// Mitsubishi GX Works2 project: GLED-3K680-20090012_210325   PLC: FX3U/FX3UC
// SECS

PROGRAM MAIN
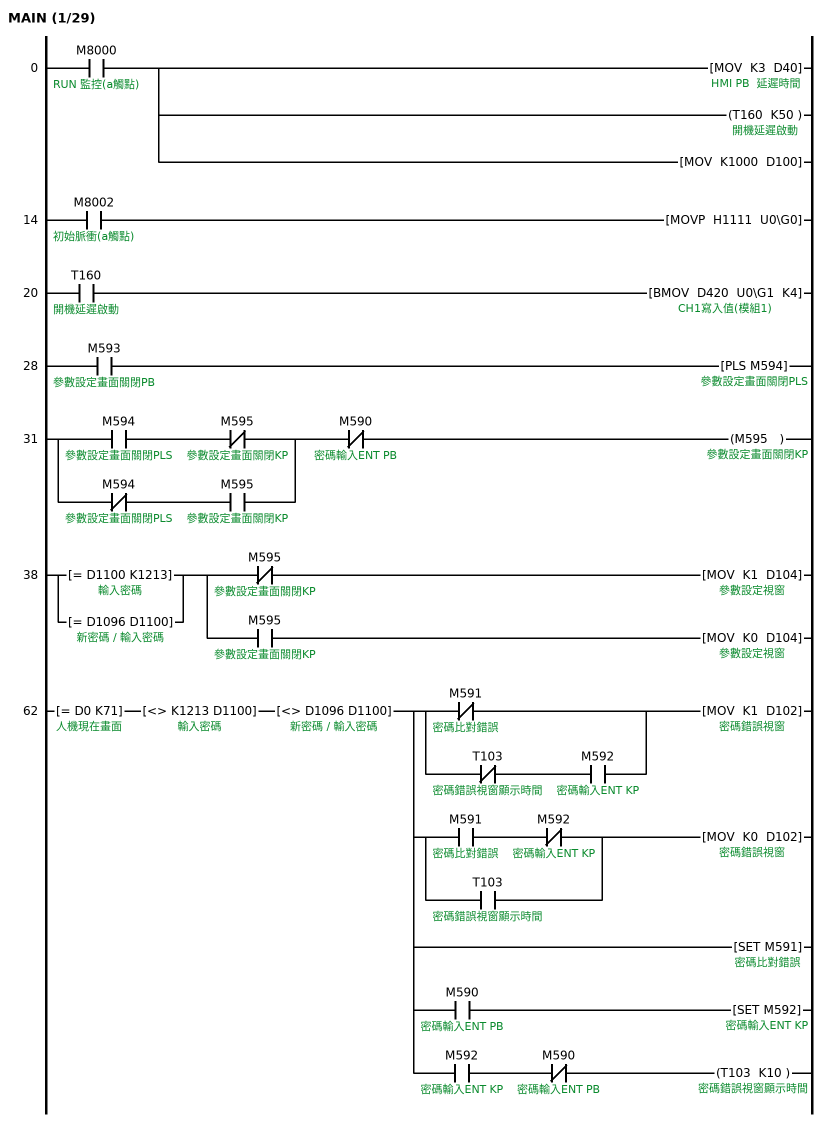
0     LD      M8000  ; RUN 監控(a觸點)
      MOV     K3 D40  ; HMI PB  延遲時間
      OUT     T160 K50  ; 開機延遲啟動
      MOV     K1000 D100
14    LD      M8002  ; 初始脈衝(a觸點)
      MOVP    H1111 U0\G0
20    LD      T160  ; 開機延遲啟動
      BMOV    D420 U0\G1 K4  ; CH1寫入值(模組1)
28    LD      M593  ; 參數設定畫面關閉PB
      PLS     M594  ; 參數設定畫面關閉PLS
31    LD      M594  ; 參數設定畫面關閉PLS
      ANI     M595  ; 參數設定畫面關閉KP
      LDI     M594  ; 參數設定畫面關閉PLS
      AND     M595  ; 參數設定畫面關閉KP
      ORB
      ANI     M590  ; 密碼輸入ENT PB
      OUT     M595  ; 參數設定畫面關閉KP
38    LD=     D1100 K1213  ; 輸入密碼
      OR=     D1096 D1100  ; 新密碼 / 輸入密碼
      MPS
      ANI     M595  ; 參數設定畫面關閉KP
      MOV     K1 D104  ; 參數設定視窗
      MPP
      AND     M595  ; 參數設定畫面關閉KP
      MOV     K0 D104
62    LD=     D0 K71  ; 人機現在畫面
      AND<>   K1213 D1100  ; 輸入密碼
      AND<>   D1096 D1100  ; 新密碼 / 輸入密碼
      MPS
      LDI     M591  ; 密碼比對錯誤
      LDI     T103  ; 密碼錯誤視窗顯示時間
      AND     M592  ; 密碼輸入ENT KP
      ORB
      ANB
      MOV     K1 D102  ; 密碼錯誤視窗
      MRD
      LD      M591  ; 密碼比對錯誤
      ANI     M592  ; 密碼輸入ENT KP
      OR      T103  ; 密碼錯誤視窗顯示時間
      ANB
      MOV     K0 D102
      MPP
      SET     M591  ; 密碼比對錯誤
      MPS
      AND     M590  ; 密碼輸入ENT PB
      SET     M592  ; 密碼輸入ENT KP
      MPP
      AND     M592  ; 密碼輸入ENT KP
      ANI     M590  ; 密碼輸入ENT PB
      OUT     T103 K10  ; 密碼錯誤視窗顯示時間
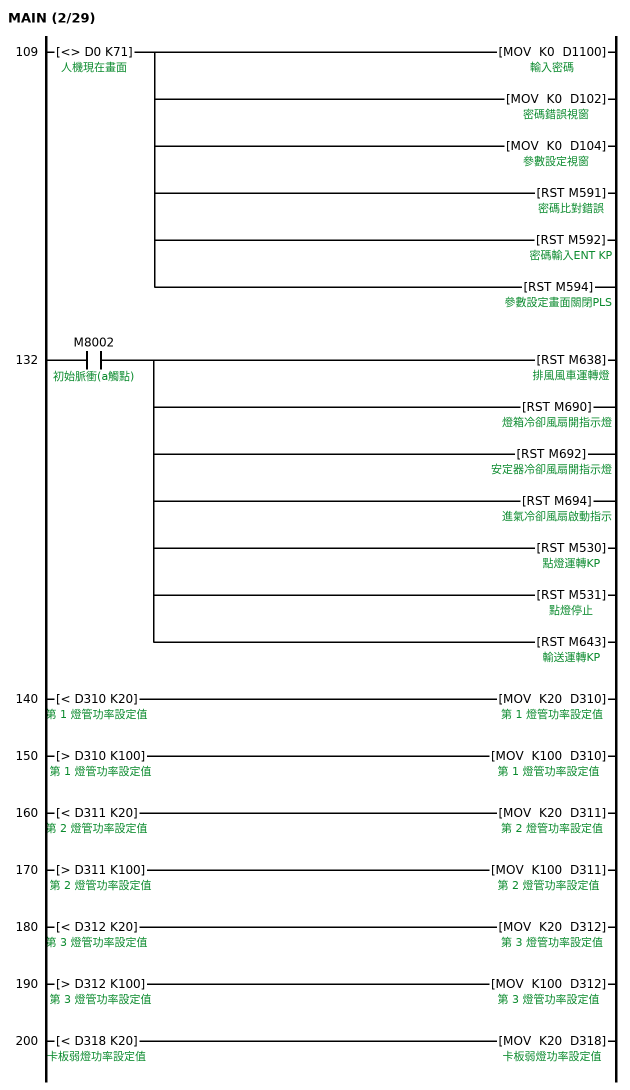
109   LD<>    D0 K71  ; 人機現在畫面
      MOV     K0 D1100
      MOV     K0 D102
      MOV     K0 D104
      RST     M591  ; 密碼比對錯誤
      RST     M592  ; 密碼輸入ENT KP
      RST     M594  ; 參數設定畫面關閉PLS
132   LD      M8002  ; 初始脈衝(a觸點)
      RST     M638  ; 排風風車運轉燈
      RST     M690  ; 燈箱冷卻風扇開指示燈
      RST     M692  ; 安定器冷卻風扇開指示燈
      RST     M694  ; 進氣冷卻風扇啟動指示
      RST     M530  ; 點燈運轉KP
      RST     M531  ; 點燈停止
      RST     M643  ; 輸送運轉KP
140   LD<     D310 K20  ; 第 1 燈管功率設定值
      MOV     K20 D310
150   LD>     D310 K100  ; 第 1 燈管功率設定值
      MOV     K100 D310
160   LD<     D311 K20  ; 第 2 燈管功率設定值
      MOV     K20 D311
170   LD>     D311 K100  ; 第 2 燈管功率設定值
      MOV     K100 D311
180   LD<     D312 K20  ; 第 3 燈管功率設定值
      MOV     K20 D312
190   LD>     D312 K100  ; 第 3 燈管功率設定值
      MOV     K100 D312
200   LD<     D318 K20  ; 卡板弱燈功率設定值
      MOV     K20 D318
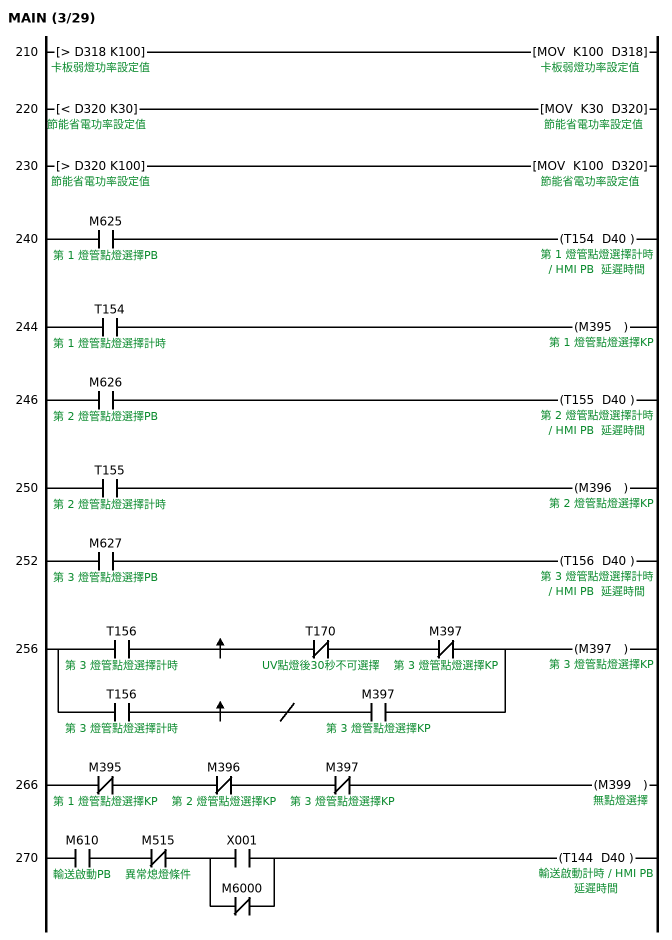
210   LD>     D318 K100  ; 卡板弱燈功率設定值
      MOV     K100 D318
220   LD<     D320 K30  ; 節能省電功率設定值
      MOV     K30 D320
230   LD>     D320 K100  ; 節能省電功率設定值
      MOV     K100 D320
240   LD      M625  ; 第 1 燈管點燈選擇PB
      OUT     T154 D40  ; 第 1 燈管點燈選擇計時 / HMI PB  延遲時間
244   LD      T154  ; 第 1 燈管點燈選擇計時
      OUT     M395  ; 第 1 燈管點燈選擇KP
246   LD      M626  ; 第 2 燈管點燈選擇PB
      OUT     T155 D40  ; 第 2 燈管點燈選擇計時 / HMI PB  延遲時間
250   LD      T155  ; 第 2 燈管點燈選擇計時
      OUT     M396  ; 第 2 燈管點燈選擇KP
252   LD      M627  ; 第 3 燈管點燈選擇PB
      OUT     T156 D40  ; 第 3 燈管點燈選擇計時 / HMI PB  延遲時間
256   LD      T156  ; 第 3 燈管點燈選擇計時
      MEP
      ANI     T170  ; UV點燈後30秒不可選擇
      ANI     M397  ; 第 3 燈管點燈選擇KP
      LD      T156  ; 第 3 燈管點燈選擇計時
      MEP
      INV
      AND     M397  ; 第 3 燈管點燈選擇KP
      ORB
      OUT     M397  ; 第 3 燈管點燈選擇KP
266   LDI     M395  ; 第 1 燈管點燈選擇KP
      ANI     M396  ; 第 2 燈管點燈選擇KP
      ANI     M397  ; 第 3 燈管點燈選擇KP
      OUT     M399  ; 無點燈選擇
270   LD      M610  ; 輸送啟動PB
      ANI     M515  ; 異常熄燈條件
      LD      X001
      ORI     M6000
      ANB
      OUT     T144 D40  ; 輸送啟動計時 / HMI PB  延遲時間
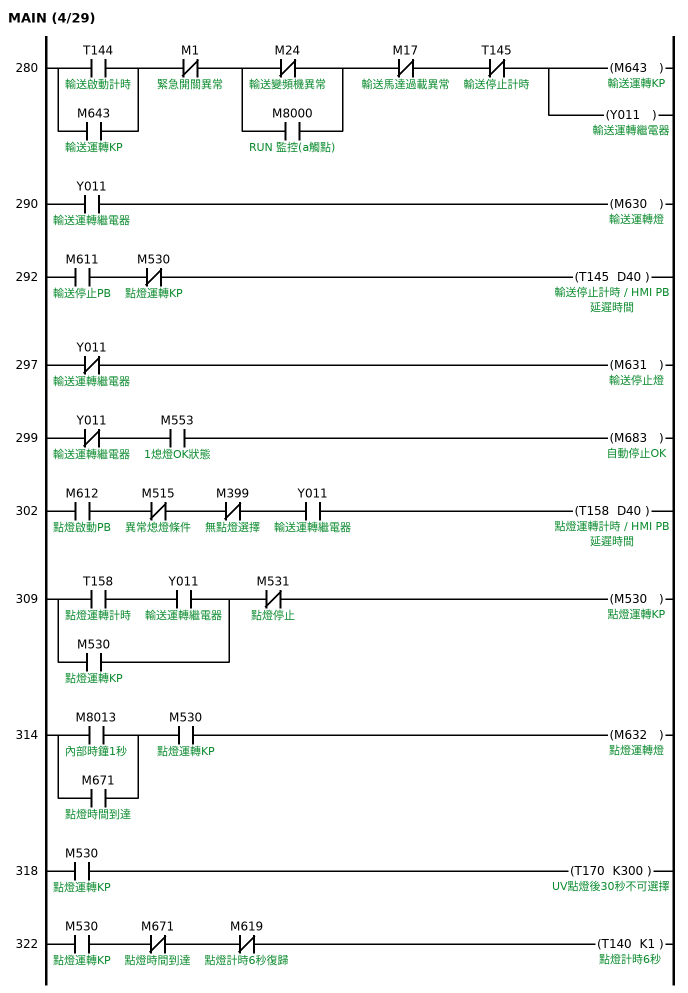
280   LD      T144  ; 輸送啟動計時
      OR      M643  ; 輸送運轉KP
      ANI     M1  ; 緊急開關異常
      LDI     M24  ; 輸送變頻機異常
      OR      M8000  ; RUN 監控(a觸點)
      ANB
      ANI     M17  ; 輸送馬達過載異常
      ANI     T145  ; 輸送停止計時
      OUT     M643  ; 輸送運轉KP
      OUT     Y011  ; 輸送運轉繼電器
290   LD      Y011  ; 輸送運轉繼電器
      OUT     M630  ; 輸送運轉燈
292   LD      M611  ; 輸送停止PB
      ANI     M530  ; 點燈運轉KP
      OUT     T145 D40  ; 輸送停止計時 / HMI PB  延遲時間
297   LDI     Y011  ; 輸送運轉繼電器
      OUT     M631  ; 輸送停止燈
299   LDI     Y011  ; 輸送運轉繼電器
      AND     M553  ; 1熄燈OK狀態
      OUT     M683  ; 自動停止OK
302   LD      M612  ; 點燈啟動PB
      ANI     M515  ; 異常熄燈條件
      ANI     M399  ; 無點燈選擇
      AND     Y011  ; 輸送運轉繼電器
      OUT     T158 D40  ; 點燈運轉計時 / HMI PB  延遲時間
309   LD      T158  ; 點燈運轉計時
      AND     Y011  ; 輸送運轉繼電器
      OR      M530  ; 點燈運轉KP
      ANI     M531  ; 點燈停止
      OUT     M530  ; 點燈運轉KP
314   LD      M8013  ; 內部時鐘1秒
      OR      M671  ; 點燈時間到達
      AND     M530  ; 點燈運轉KP
      OUT     M632  ; 點燈運轉燈
318   LD      M530  ; 點燈運轉KP
      OUT     T170 K300  ; UV點燈後30秒不可選擇
322   LD      M530  ; 點燈運轉KP
      ANI     M671  ; 點燈時間到達
      ANI     M619  ; 點燈計時6秒復歸
      OUT     T140 K1  ; 點燈計時6秒
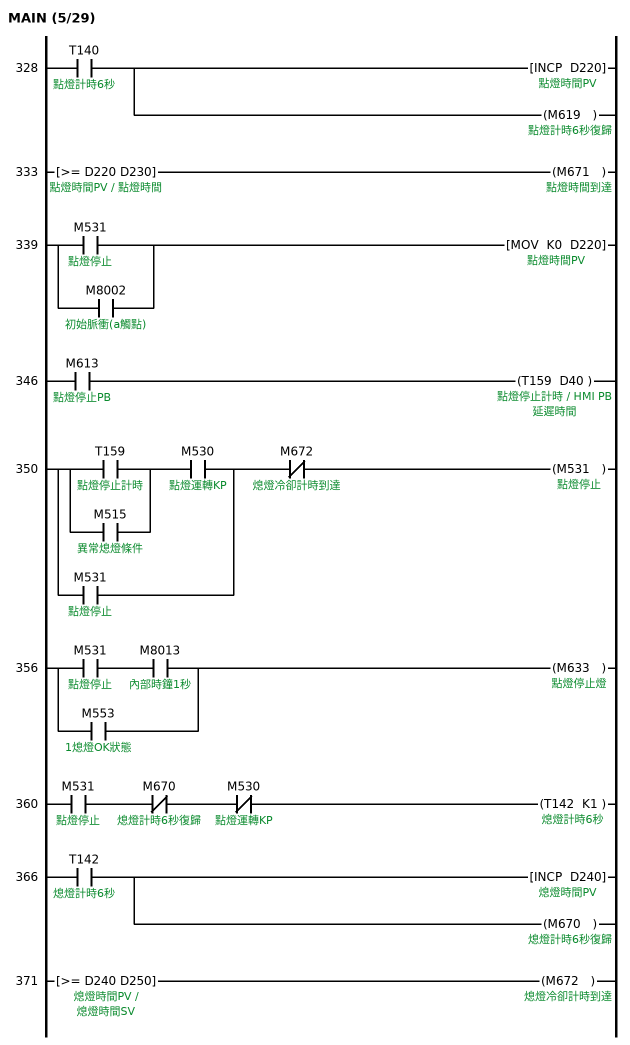
328   LD      T140  ; 點燈計時6秒
      INCP    D220  ; 點燈時間PV
      OUT     M619  ; 點燈計時6秒復歸
333   LD>=    D220 D230  ; 點燈時間PV / 點燈時間
      OUT     M671  ; 點燈時間到達
339   LD      M531  ; 點燈停止
      OR      M8002  ; 初始脈衝(a觸點)
      MOV     K0 D220
346   LD      M613  ; 點燈停止PB
      OUT     T159 D40  ; 點燈停止計時 / HMI PB  延遲時間
350   LD      T159  ; 點燈停止計時
      OR      M515  ; 異常熄燈條件
      AND     M530  ; 點燈運轉KP
      OR      M531  ; 點燈停止
      ANI     M672  ; 熄燈冷卻計時到達
      OUT     M531  ; 點燈停止
356   LD      M531  ; 點燈停止
      AND     M8013  ; 內部時鐘1秒
      OR      M553  ; 1熄燈OK狀態
      OUT     M633  ; 點燈停止燈
360   LD      M531  ; 點燈停止
      ANI     M670  ; 熄燈計時6秒復歸
      ANI     M530  ; 點燈運轉KP
      OUT     T142 K1  ; 熄燈計時6秒
366   LD      T142  ; 熄燈計時6秒
      INCP    D240  ; 熄燈時間PV
      OUT     M670  ; 熄燈計時6秒復歸
371   LD>=    D240 D250  ; 熄燈時間PV / 熄燈時間SV
      OUT     M672  ; 熄燈冷卻計時到達
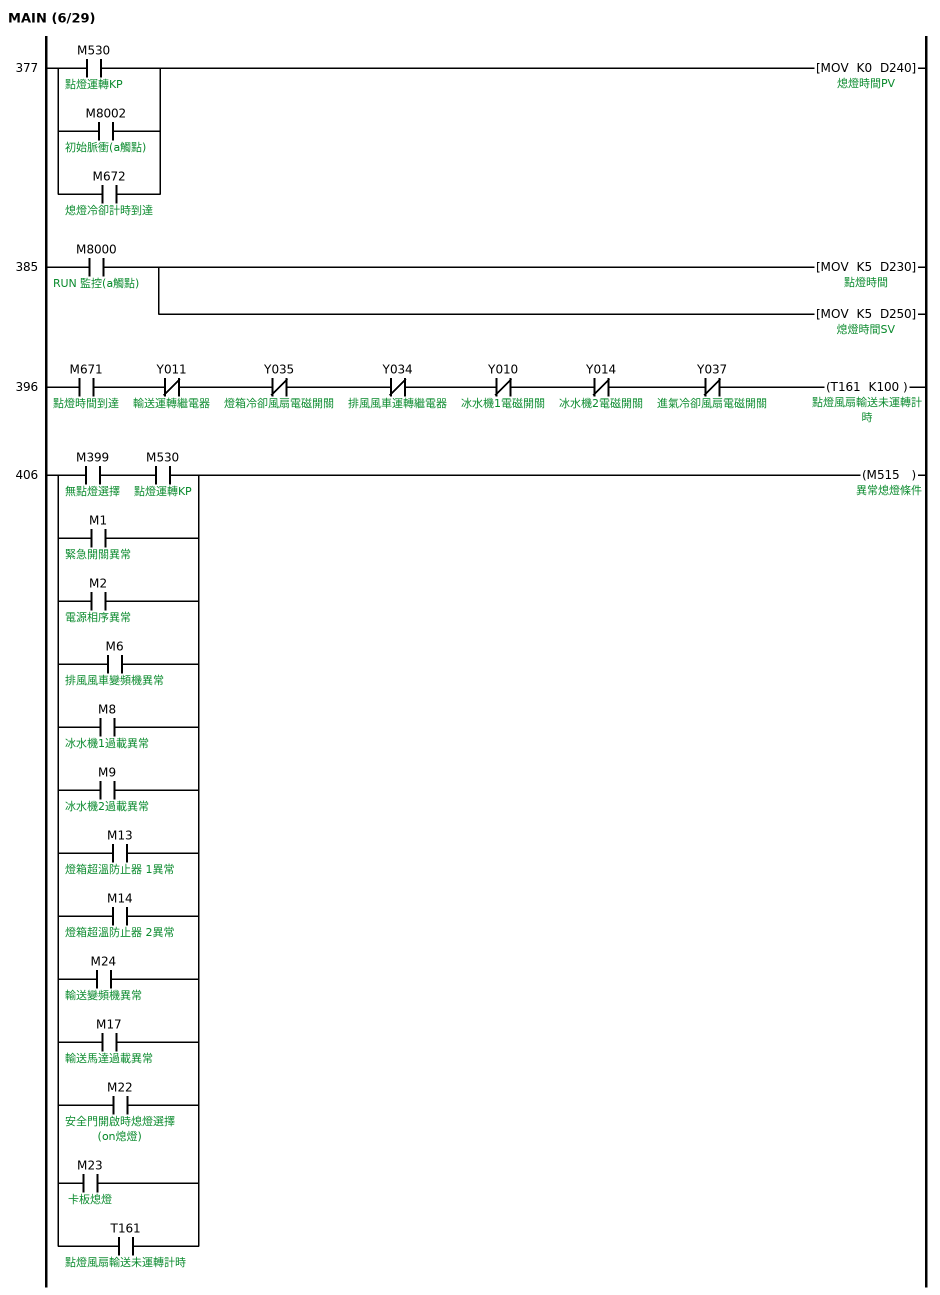
377   LD      M530  ; 點燈運轉KP
      OR      M8002  ; 初始脈衝(a觸點)
      OR      M672  ; 熄燈冷卻計時到達
      MOV     K0 D240
385   LD      M8000  ; RUN 監控(a觸點)
      MOV     K5 D230
      MOV     K5 D250
396   LD      M671  ; 點燈時間到達
      ANI     Y011  ; 輸送運轉繼電器
      ANI     Y035  ; 燈箱冷卻風扇電磁開關
      ANI     Y034  ; 排風風車運轉繼電器
      ANI     Y010  ; 冰水機1電磁開關
      ANI     Y014  ; 冰水機2電磁開關
      ANI     Y037  ; 進氣冷卻風扇電磁開關
      OUT     T161 K100  ; 點燈風扇輸送未運轉計時
406   LD      M399  ; 無點燈選擇
      AND     M530  ; 點燈運轉KP
      OR      M1  ; 緊急開關異常
      OR      M2  ; 電源相序異常
      OR      M6  ; 排風風車變頻機異常
      OR      M8  ; 冰水機1過載異常
      OR      M9  ; 冰水機2過載異常
      OR      M13  ; 燈箱超溫防止器 1異常
      OR      M14  ; 燈箱超溫防止器 2異常
      OR      M24  ; 輸送變頻機異常
      OR      M17  ; 輸送馬達過載異常
      OR      M22  ; 安全門開啟時熄燈選擇    (on熄燈)
      OR      M23  ; 卡板熄燈
      OR      T161  ; 點燈風扇輸送未運轉計時
      OUT     M515  ; 異常熄燈條件
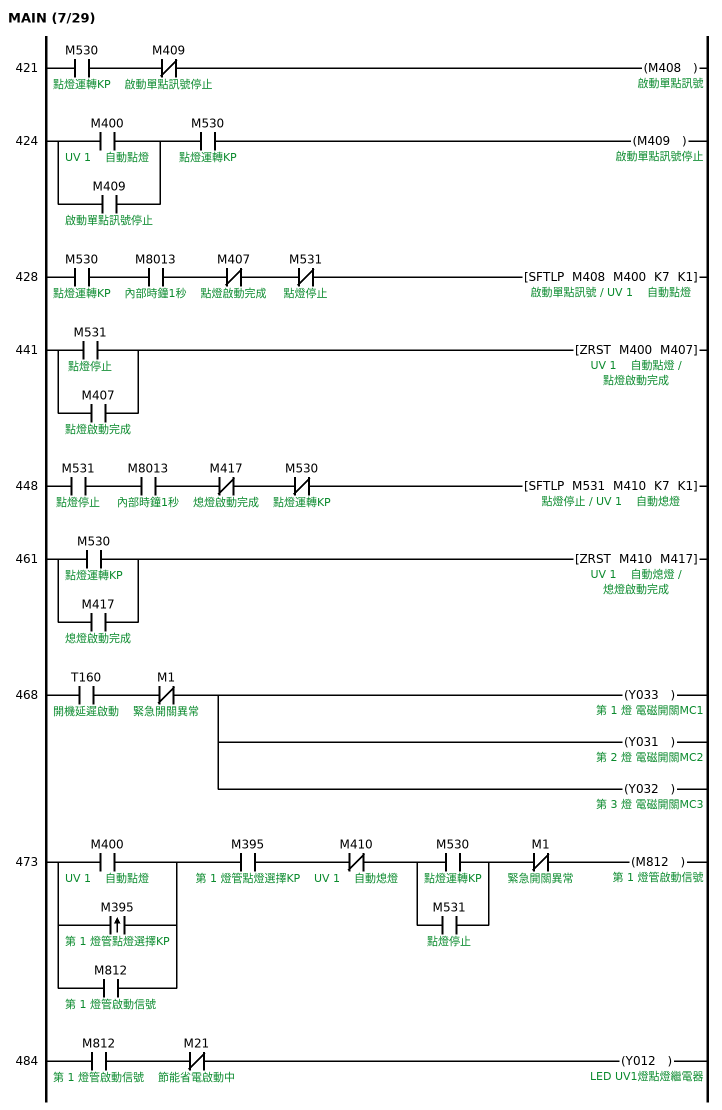
421   LD      M530  ; 點燈運轉KP
      ANI     M409  ; 啟動單點訊號停止
      OUT     M408  ; 啟動單點訊號
424   LD      M400  ; UV 1    自動點燈
      OR      M409  ; 啟動單點訊號停止
      AND     M530  ; 點燈運轉KP
      OUT     M409  ; 啟動單點訊號停止
428   LD      M530  ; 點燈運轉KP
      AND     M8013  ; 內部時鐘1秒
      ANI     M407  ; 點燈啟動完成
      ANI     M531  ; 點燈停止
      SFTLP   M408 M400 K7 K1
441   LD      M531  ; 點燈停止
      OR      M407  ; 點燈啟動完成
      ZRST    M400 M407
448   LD      M531  ; 點燈停止
      AND     M8013  ; 內部時鐘1秒
      ANI     M417  ; 熄燈啟動完成
      ANI     M530  ; 點燈運轉KP
      SFTLP   M531 M410 K7 K1  ; UV 1    自動熄燈
461   LD      M530  ; 點燈運轉KP
      OR      M417  ; 熄燈啟動完成
      ZRST    M410 M417
468   LD      T160  ; 開機延遲啟動
      ANI     M1  ; 緊急開關異常
      OUT     Y033  ; 第 1 燈 電磁開關MC1
      OUT     Y031  ; 第 2 燈 電磁開關MC2
      OUT     Y032  ; 第 3 燈 電磁開關MC3
473   LD      M400  ; UV 1    自動點燈
      ORP     M395  ; 第 1 燈管點燈選擇KP
      OR      M812  ; 第 1 燈管啟動信號
      AND     M395  ; 第 1 燈管點燈選擇KP
      ANI     M410  ; UV 1    自動熄燈
      LD      M530  ; 點燈運轉KP
      OR      M531  ; 點燈停止
      ANB
      ANI     M1  ; 緊急開關異常
      OUT     M812  ; 第 1 燈管啟動信號
484   LD      M812  ; 第 1 燈管啟動信號
      ANI     M21  ; 節能省電啟動中
      OUT     Y012  ; LED UV1燈點燈繼電器
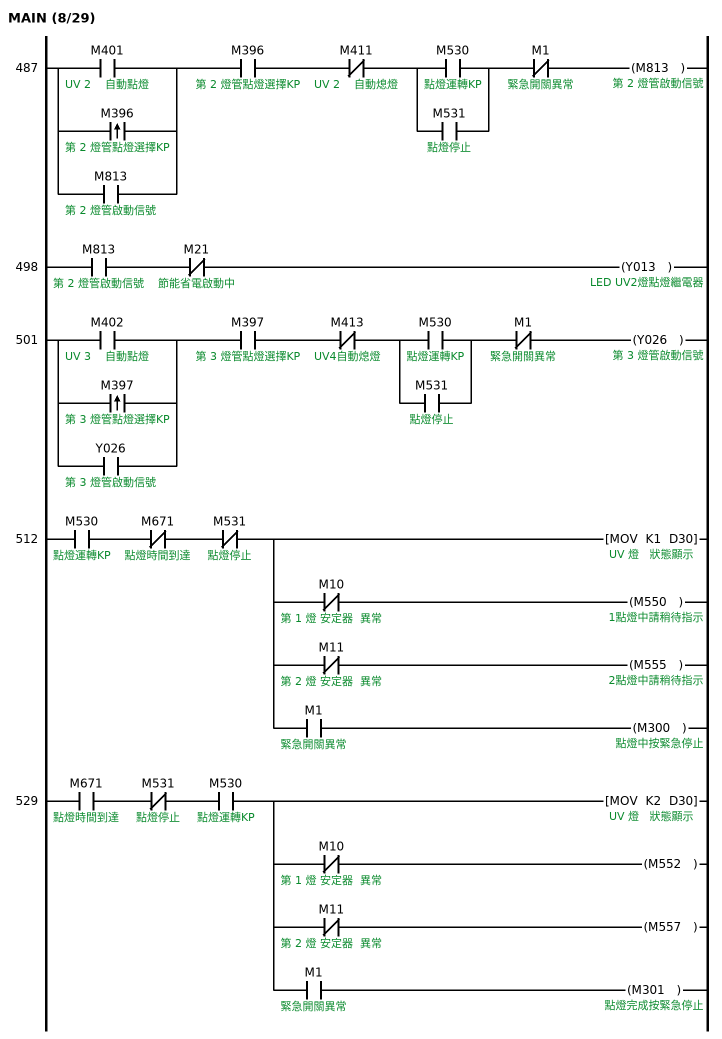
487   LD      M401  ; UV 2    自動點燈
      ORP     M396  ; 第 2 燈管點燈選擇KP
      OR      M813  ; 第 2 燈管啟動信號
      AND     M396  ; 第 2 燈管點燈選擇KP
      ANI     M411  ; UV 2    自動熄燈
      LD      M530  ; 點燈運轉KP
      OR      M531  ; 點燈停止
      ANB
      ANI     M1  ; 緊急開關異常
      OUT     M813  ; 第 2 燈管啟動信號
498   LD      M813  ; 第 2 燈管啟動信號
      ANI     M21  ; 節能省電啟動中
      OUT     Y013  ; LED UV2燈點燈繼電器
501   LD      M402  ; UV 3    自動點燈
      ORP     M397  ; 第 3 燈管點燈選擇KP
      OR      Y026  ; 第 3 燈管啟動信號
      AND     M397  ; 第 3 燈管點燈選擇KP
      ANI     M413  ; UV4自動熄燈
      LD      M530  ; 點燈運轉KP
      OR      M531  ; 點燈停止
      ANB
      ANI     M1  ; 緊急開關異常
      OUT     Y026  ; 第 3 燈管啟動信號
512   LD      M530  ; 點燈運轉KP
      ANI     M671  ; 點燈時間到達
      ANI     M531  ; 點燈停止
      MOV     K1 D30  ; UV 燈   狀態顯示
      MPS
      ANI     M10  ; 第 1 燈 安定器  異常
      OUT     M550  ; 1點燈中請稍待指示
      MRD
      ANI     M11  ; 第 2 燈 安定器  異常
      OUT     M555  ; 2點燈中請稍待指示
      MPP
      AND     M1  ; 緊急開關異常
      OUT     M300  ; 點燈中按緊急停止
529   LD      M671  ; 點燈時間到達
      ANI     M531  ; 點燈停止
      AND     M530  ; 點燈運轉KP
      MOV     K2 D30
      MPS
      ANI     M10  ; 第 1 燈 安定器  異常
      OUT     M552
      MRD
      ANI     M11  ; 第 2 燈 安定器  異常
      OUT     M557
      MPP
      AND     M1  ; 緊急開關異常
      OUT     M301  ; 點燈完成按緊急停止
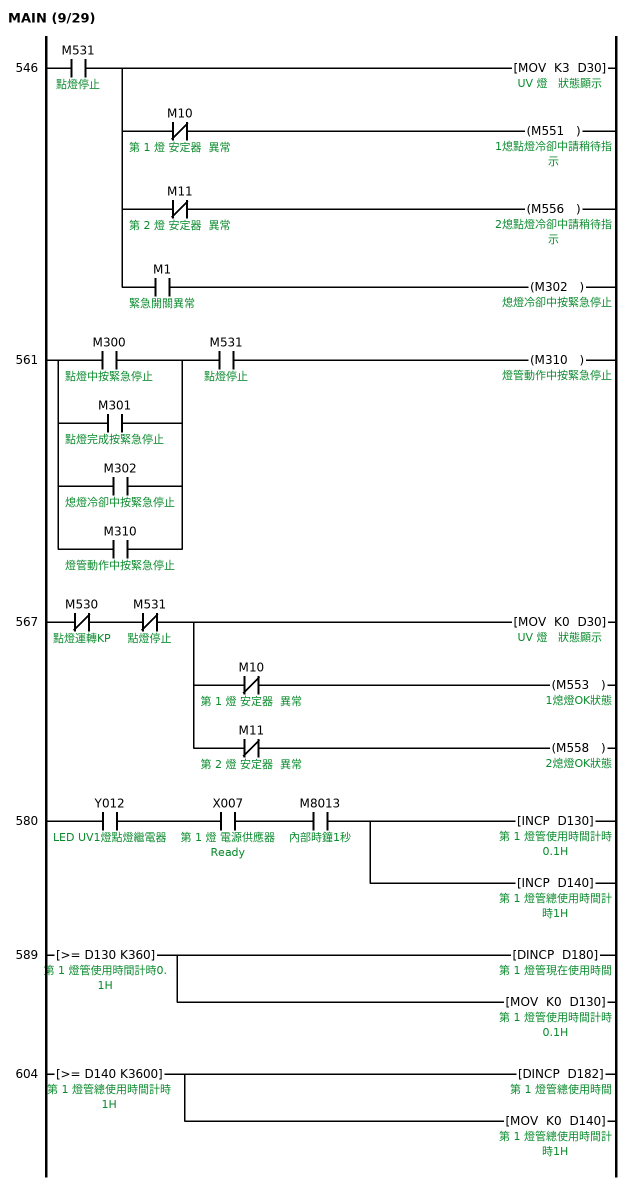
546   LD      M531  ; 點燈停止
      MOV     K3 D30
      MPS
      ANI     M10  ; 第 1 燈 安定器  異常
      OUT     M551  ; 1熄點燈冷卻中請稍待指示
      MRD
      ANI     M11  ; 第 2 燈 安定器  異常
      OUT     M556  ; 2熄點燈冷卻中請稍待指示
      MPP
      AND     M1  ; 緊急開關異常
      OUT     M302  ; 熄燈冷卻中按緊急停止
561   LD      M300  ; 點燈中按緊急停止
      OR      M301  ; 點燈完成按緊急停止
      OR      M302  ; 熄燈冷卻中按緊急停止
      OR      M310  ; 燈管動作中按緊急停止
      AND     M531  ; 點燈停止
      OUT     M310  ; 燈管動作中按緊急停止
567   LDI     M530  ; 點燈運轉KP
      ANI     M531  ; 點燈停止
      MOV     K0 D30
      MPS
      ANI     M10  ; 第 1 燈 安定器  異常
      OUT     M553  ; 1熄燈OK狀態
      MPP
      ANI     M11  ; 第 2 燈 安定器  異常
      OUT     M558  ; 2熄燈OK狀態
580   LD      Y012  ; LED UV1燈點燈繼電器
      AND     X007  ; 第 1 燈 電源供應器 Ready
      AND     M8013  ; 內部時鐘1秒
      INCP    D130  ; 第 1 燈管使用時間計時0.1H
      INCP    D140  ; 第 1 燈管總使用時間計時1H
589   LD>=    D130 K360  ; 第 1 燈管使用時間計時0.1H
      DINCP   D180  ; 第 1 燈管現在使用時間
      MOV     K0 D130
604   LD>=    D140 K3600  ; 第 1 燈管總使用時間計時1H
      DINCP   D182  ; 第 1 燈管總使用時間
      MOV     K0 D140
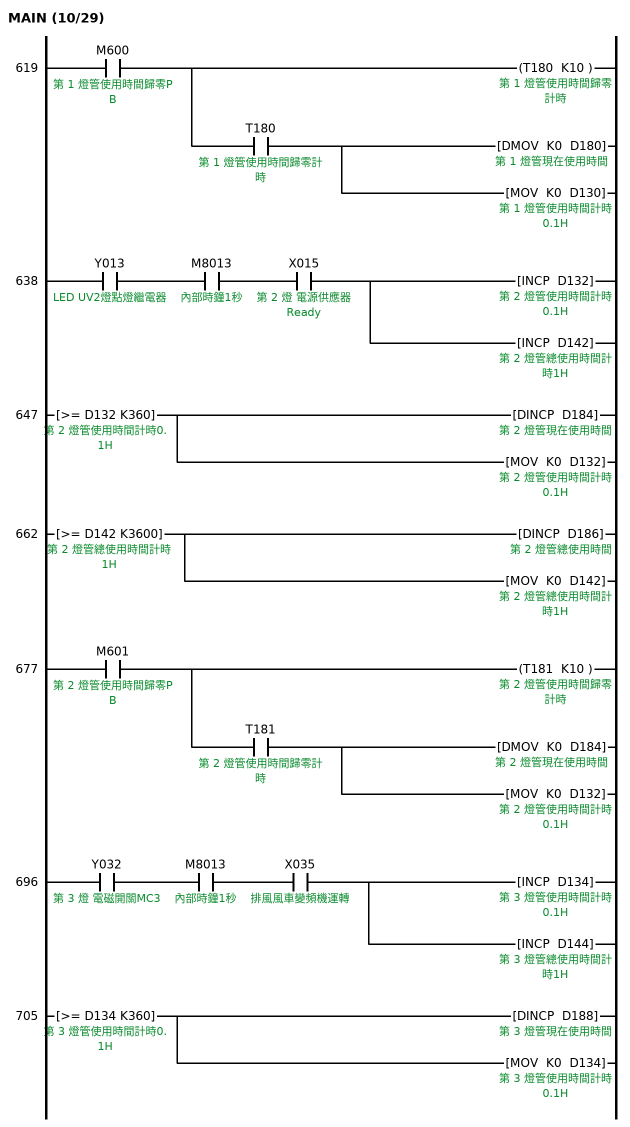
619   LD      M600  ; 第 1 燈管使用時間歸零PB
      OUT     T180 K10  ; 第 1 燈管使用時間歸零計時
      AND     T180  ; 第 1 燈管使用時間歸零計時
      DMOV    K0 D180
      MOV     K0 D130
638   LD      Y013  ; LED UV2燈點燈繼電器
      AND     M8013  ; 內部時鐘1秒
      AND     X015  ; 第 2 燈 電源供應器 Ready
      INCP    D132  ; 第 2 燈管使用時間計時0.1H
      INCP    D142  ; 第 2 燈管總使用時間計時1H
647   LD>=    D132 K360  ; 第 2 燈管使用時間計時0.1H
      DINCP   D184  ; 第 2 燈管現在使用時間
      MOV     K0 D132
662   LD>=    D142 K3600  ; 第 2 燈管總使用時間計時1H
      DINCP   D186  ; 第 2 燈管總使用時間
      MOV     K0 D142
677   LD      M601  ; 第 2 燈管使用時間歸零PB
      OUT     T181 K10  ; 第 2 燈管使用時間歸零計時
      AND     T181  ; 第 2 燈管使用時間歸零計時
      DMOV    K0 D184
      MOV     K0 D132
696   LD      Y032  ; 第 3 燈 電磁開關MC3
      AND     M8013  ; 內部時鐘1秒
      AND     X035  ; 排風風車變頻機運轉
      INCP    D134  ; 第 3 燈管使用時間計時0.1H
      INCP    D144  ; 第 3 燈管總使用時間計時1H
705   LD>=    D134 K360  ; 第 3 燈管使用時間計時0.1H
      DINCP   D188  ; 第 3 燈管現在使用時間
      MOV     K0 D134
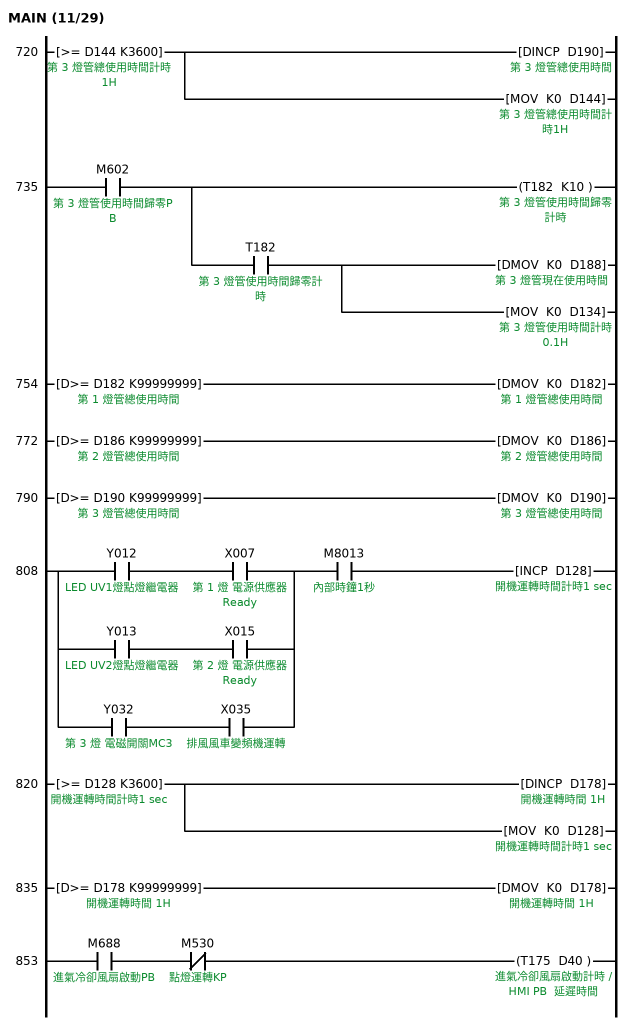
720   LD>=    D144 K3600  ; 第 3 燈管總使用時間計時1H
      DINCP   D190  ; 第 3 燈管總使用時間
      MOV     K0 D144
735   LD      M602  ; 第 3 燈管使用時間歸零PB
      OUT     T182 K10  ; 第 3 燈管使用時間歸零計時
      AND     T182  ; 第 3 燈管使用時間歸零計時
      DMOV    K0 D188
      MOV     K0 D134
754   LDD>=   D182 K99999999  ; 第 1 燈管總使用時間
      DMOV    K0 D182
772   LDD>=   D186 K99999999  ; 第 2 燈管總使用時間
      DMOV    K0 D186
790   LDD>=   D190 K99999999  ; 第 3 燈管總使用時間
      DMOV    K0 D190
808   LD      Y012  ; LED UV1燈點燈繼電器
      AND     X007  ; 第 1 燈 電源供應器 Ready
      LD      Y013  ; LED UV2燈點燈繼電器
      AND     X015  ; 第 2 燈 電源供應器 Ready
      ORB
      LD      Y032  ; 第 3 燈 電磁開關MC3
      AND     X035  ; 排風風車變頻機運轉
      ORB
      AND     M8013  ; 內部時鐘1秒
      INCP    D128  ; 開機運轉時間計時1 sec
820   LD>=    D128 K3600  ; 開機運轉時間計時1 sec
      DINCP   D178  ; 開機運轉時間 1H
      MOV     K0 D128
835   LDD>=   D178 K99999999  ; 開機運轉時間 1H
      DMOV    K0 D178
853   LD      M688  ; 進氣冷卻風扇啟動PB
      ANI     M530  ; 點燈運轉KP
      OUT     T175 D40  ; 進氣冷卻風扇啟動計時 / HMI PB  延遲時間
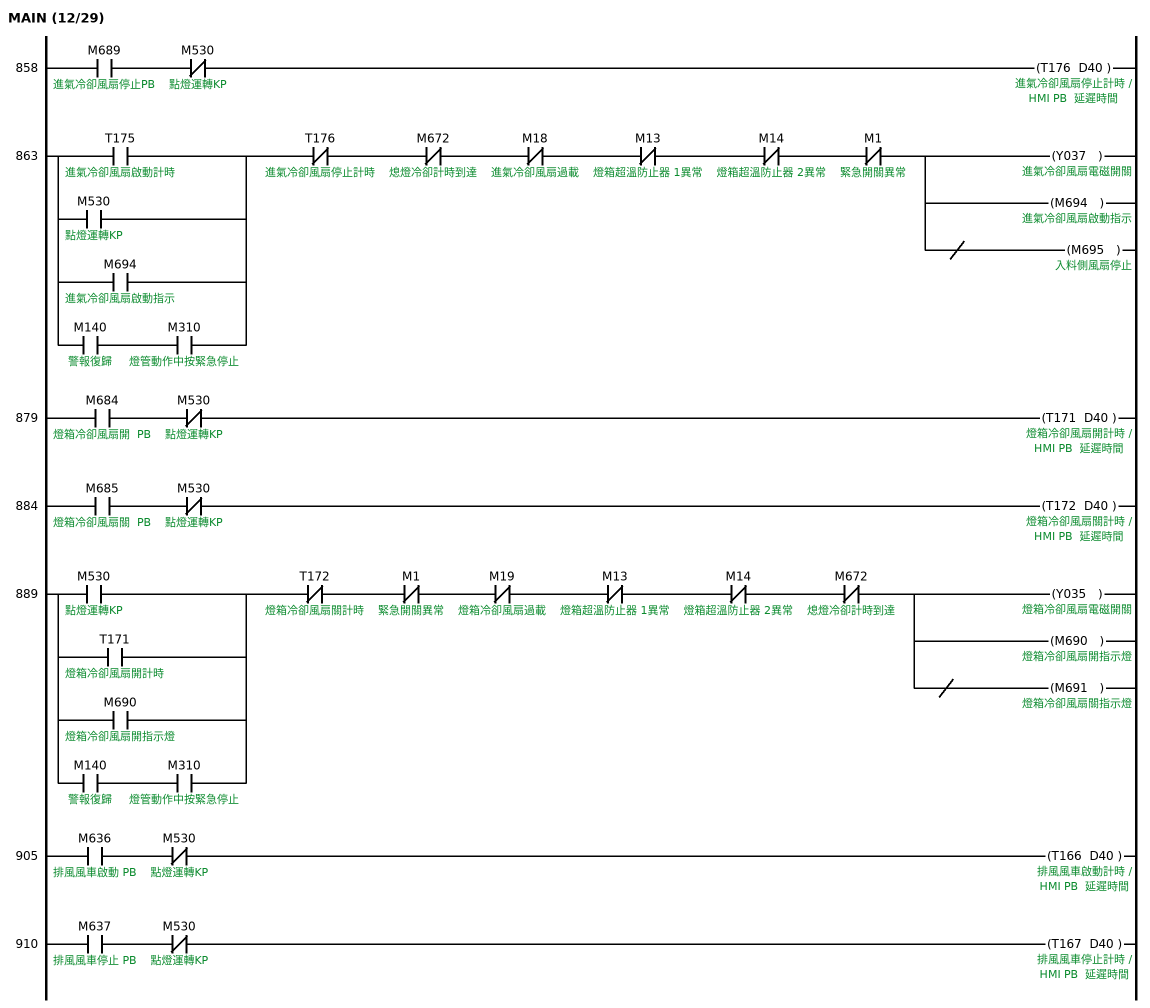
858   LD      M689  ; 進氣冷卻風扇停止PB
      ANI     M530  ; 點燈運轉KP
      OUT     T176 D40  ; 進氣冷卻風扇停止計時 / HMI PB  延遲時間
863   LD      T175  ; 進氣冷卻風扇啟動計時
      OR      M530  ; 點燈運轉KP
      OR      M694  ; 進氣冷卻風扇啟動指示
      LD      M140  ; 警報復歸
      AND     M310  ; 燈管動作中按緊急停止
      ORB
      ANI     T176  ; 進氣冷卻風扇停止計時
      ANI     M672  ; 熄燈冷卻計時到達
      ANI     M18  ; 進氣冷卻風扇過載
      ANI     M13  ; 燈箱超溫防止器 1異常
      ANI     M14  ; 燈箱超溫防止器 2異常
      ANI     M1  ; 緊急開關異常
      OUT     Y037  ; 進氣冷卻風扇電磁開關
      OUT     M694  ; 進氣冷卻風扇啟動指示
      INV
      OUT     M695  ; 入料側風扇停止
879   LD      M684  ; 燈箱冷卻風扇開  PB
      ANI     M530  ; 點燈運轉KP
      OUT     T171 D40  ; 燈箱冷卻風扇開計時 / HMI PB  延遲時間
884   LD      M685  ; 燈箱冷卻風扇關  PB
      ANI     M530  ; 點燈運轉KP
      OUT     T172 D40  ; 燈箱冷卻風扇關計時 / HMI PB  延遲時間
889   LD      M530  ; 點燈運轉KP
      OR      T171  ; 燈箱冷卻風扇開計時
      OR      M690  ; 燈箱冷卻風扇開指示燈
      LD      M140  ; 警報復歸
      AND     M310  ; 燈管動作中按緊急停止
      ORB
      ANI     T172  ; 燈箱冷卻風扇關計時
      ANI     M1  ; 緊急開關異常
      ANI     M19  ; 燈箱冷卻風扇過載
      ANI     M13  ; 燈箱超溫防止器 1異常
      ANI     M14  ; 燈箱超溫防止器 2異常
      ANI     M672  ; 熄燈冷卻計時到達
      OUT     Y035  ; 燈箱冷卻風扇電磁開關
      OUT     M690  ; 燈箱冷卻風扇開指示燈
      INV
      OUT     M691  ; 燈箱冷卻風扇關指示燈
905   LD      M636  ; 排風風車啟動 PB
      ANI     M530  ; 點燈運轉KP
      OUT     T166 D40  ; 排風風車啟動計時 / HMI PB  延遲時間
910   LD      M637  ; 排風風車停止 PB
      ANI     M530  ; 點燈運轉KP
      OUT     T167 D40  ; 排風風車停止計時 / HMI PB  延遲時間
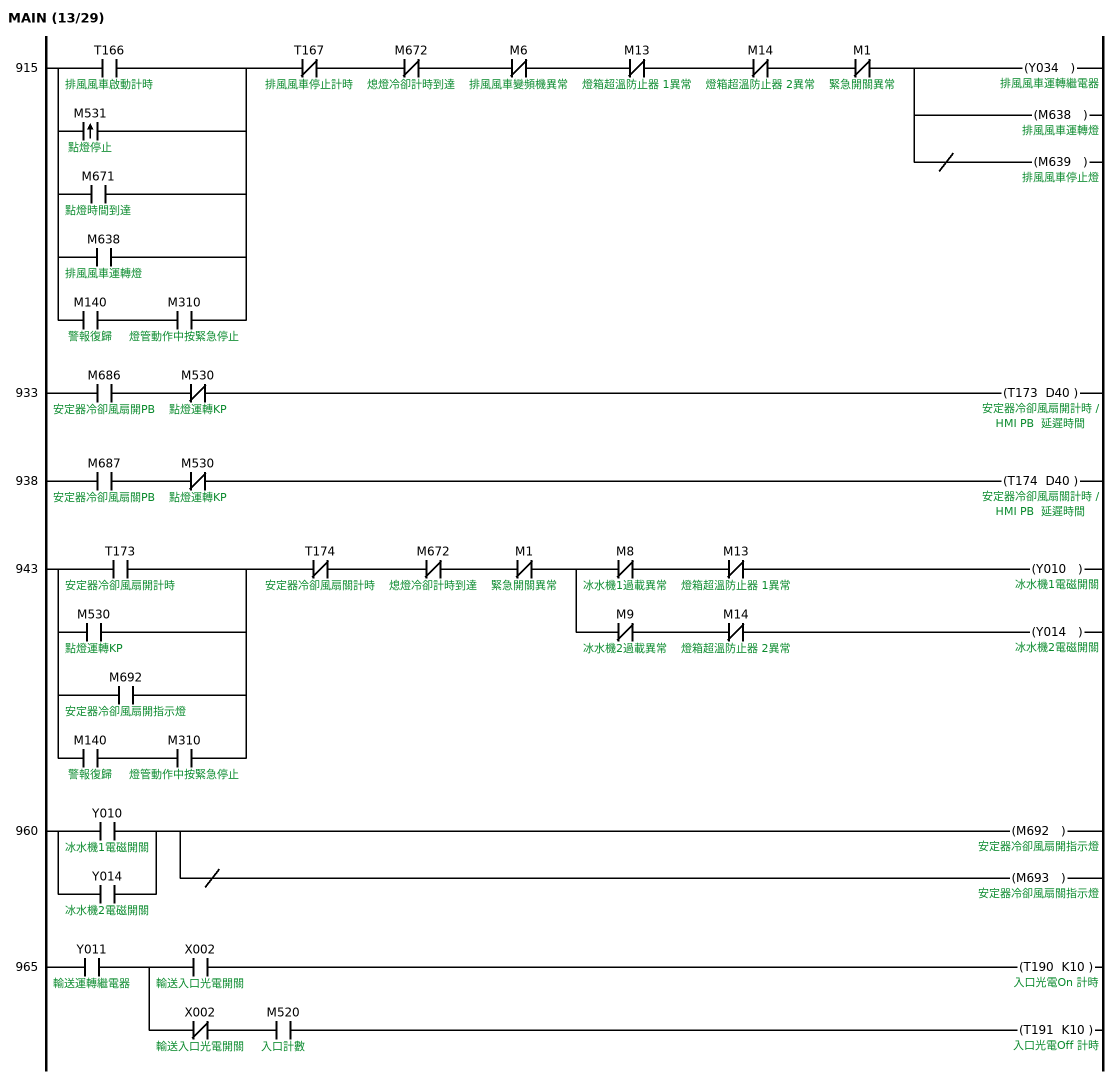
915   LD      T166  ; 排風風車啟動計時
      ORP     M531  ; 點燈停止
      OR      M671  ; 點燈時間到達
      OR      M638  ; 排風風車運轉燈
      LD      M140  ; 警報復歸
      AND     M310  ; 燈管動作中按緊急停止
      ORB
      ANI     T167  ; 排風風車停止計時
      ANI     M672  ; 熄燈冷卻計時到達
      ANI     M6  ; 排風風車變頻機異常
      ANI     M13  ; 燈箱超溫防止器 1異常
      ANI     M14  ; 燈箱超溫防止器 2異常
      ANI     M1  ; 緊急開關異常
      OUT     Y034  ; 排風風車運轉繼電器
      OUT     M638  ; 排風風車運轉燈
      INV
      OUT     M639  ; 排風風車停止燈
933   LD      M686  ; 安定器冷卻風扇開PB
      ANI     M530  ; 點燈運轉KP
      OUT     T173 D40  ; 安定器冷卻風扇開計時 / HMI PB  延遲時間
938   LD      M687  ; 安定器冷卻風扇關PB
      ANI     M530  ; 點燈運轉KP
      OUT     T174 D40  ; 安定器冷卻風扇關計時 / HMI PB  延遲時間
943   LD      T173  ; 安定器冷卻風扇開計時
      OR      M530  ; 點燈運轉KP
      OR      M692  ; 安定器冷卻風扇開指示燈
      LD      M140  ; 警報復歸
      AND     M310  ; 燈管動作中按緊急停止
      ORB
      ANI     T174  ; 安定器冷卻風扇關計時
      ANI     M672  ; 熄燈冷卻計時到達
      ANI     M1  ; 緊急開關異常
      MPS
      ANI     M8  ; 冰水機1過載異常
      ANI     M13  ; 燈箱超溫防止器 1異常
      OUT     Y010  ; 冰水機1電磁開關
      MPP
      ANI     M9  ; 冰水機2過載異常
      ANI     M14  ; 燈箱超溫防止器 2異常
      OUT     Y014  ; 冰水機2電磁開關
960   LD      Y010  ; 冰水機1電磁開關
      OR      Y014  ; 冰水機2電磁開關
      OUT     M692  ; 安定器冷卻風扇開指示燈
      INV
      OUT     M693  ; 安定器冷卻風扇關指示燈
965   LD      Y011  ; 輸送運轉繼電器
      MPS
      AND     X002  ; 輸送入口光電開關
      OUT     T190 K10  ; 入口光電On 計時
      MPP
      ANI     X002  ; 輸送入口光電開關
      AND     M520  ; 入口計數
      OUT     T191 K10  ; 入口光電Off 計時
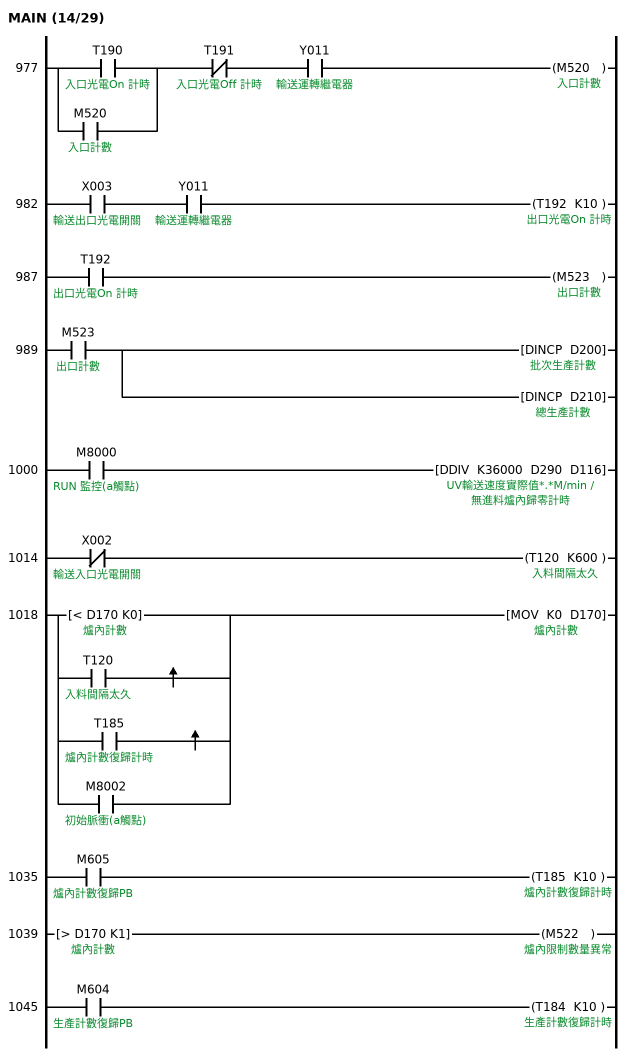
977   LD      T190  ; 入口光電On 計時
      OR      M520  ; 入口計數
      ANI     T191  ; 入口光電Off 計時
      AND     Y011  ; 輸送運轉繼電器
      OUT     M520  ; 入口計數
982   LD      X003  ; 輸送出口光電開關
      AND     Y011  ; 輸送運轉繼電器
      OUT     T192 K10  ; 出口光電On 計時
987   LD      T192  ; 出口光電On 計時
      OUT     M523  ; 出口計數
989   LD      M523  ; 出口計數
      DINCP   D200  ; 批次生產計數
      DINCP   D210  ; 總生產計數
1000  LD      M8000  ; RUN 監控(a觸點)
      DDIV    K36000 D290 D116  ; UV輸送速度實際值*.*M/min / 無進料爐內歸零計時
1014  LDI     X002  ; 輸送入口光電開關
      OUT     T120 K600  ; 入料間隔太久
1018  LD<     D170 K0  ; 爐內計數
      LD      T120  ; 入料間隔太久
      MEP
      ORB
      LD      T185  ; 爐內計數復歸計時
      MEP
      ORB
      OR      M8002  ; 初始脈衝(a觸點)
      MOV     K0 D170
1035  LD      M605  ; 爐內計數復歸PB
      OUT     T185 K10  ; 爐內計數復歸計時
1039  LD>     D170 K1  ; 爐內計數
      OUT     M522  ; 爐內限制數量異常
1045  LD      M604  ; 生產計數復歸PB
      OUT     T184 K10  ; 生產計數復歸計時
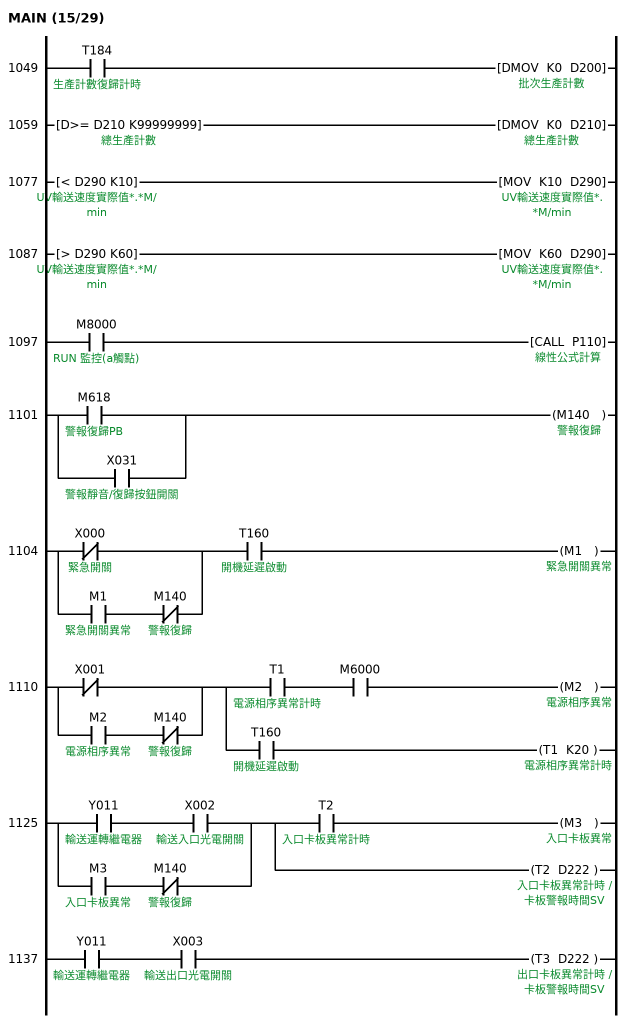
1049  LD      T184  ; 生產計數復歸計時
      DMOV    K0 D200
1059  LDD>=   D210 K99999999  ; 總生產計數
      DMOV    K0 D210
1077  LD<     D290 K10  ; UV輸送速度實際值*.*M/min
      MOV     K10 D290
1087  LD>     D290 K60  ; UV輸送速度實際值*.*M/min
      MOV     K60 D290
1097  LD      M8000  ; RUN 監控(a觸點)
      CALL    P110  ; 線性公式計算
1101  LD      M618  ; 警報復歸PB
      OR      X031  ; 警報靜音/復歸按鈕開關
      OUT     M140  ; 警報復歸
1104  LDI     X000  ; 緊急開關
      LD      M1  ; 緊急開關異常
      ANI     M140  ; 警報復歸
      ORB
      AND     T160  ; 開機延遲啟動
      OUT     M1  ; 緊急開關異常
1110  LDI     X001
      LD      M2  ; 電源相序異常
      ANI     M140  ; 警報復歸
      ORB
      MPS
      AND     T1  ; 電源相序異常計時
      AND     M6000
      OUT     M2  ; 電源相序異常
      MPP
      AND     T160  ; 開機延遲啟動
      OUT     T1 K20  ; 電源相序異常計時
1125  LD      Y011  ; 輸送運轉繼電器
      AND     X002  ; 輸送入口光電開關
      LD      M3  ; 入口卡板異常
      ANI     M140  ; 警報復歸
      ORB
      MPS
      AND     T2  ; 入口卡板異常計時
      OUT     M3  ; 入口卡板異常
      MPP
      OUT     T2 D222  ; 入口卡板異常計時 / 卡板警報時間SV
1137  LD      Y011  ; 輸送運轉繼電器
      AND     X003  ; 輸送出口光電開關
      OUT     T3 D222  ; 出口卡板異常計時 / 卡板警報時間SV
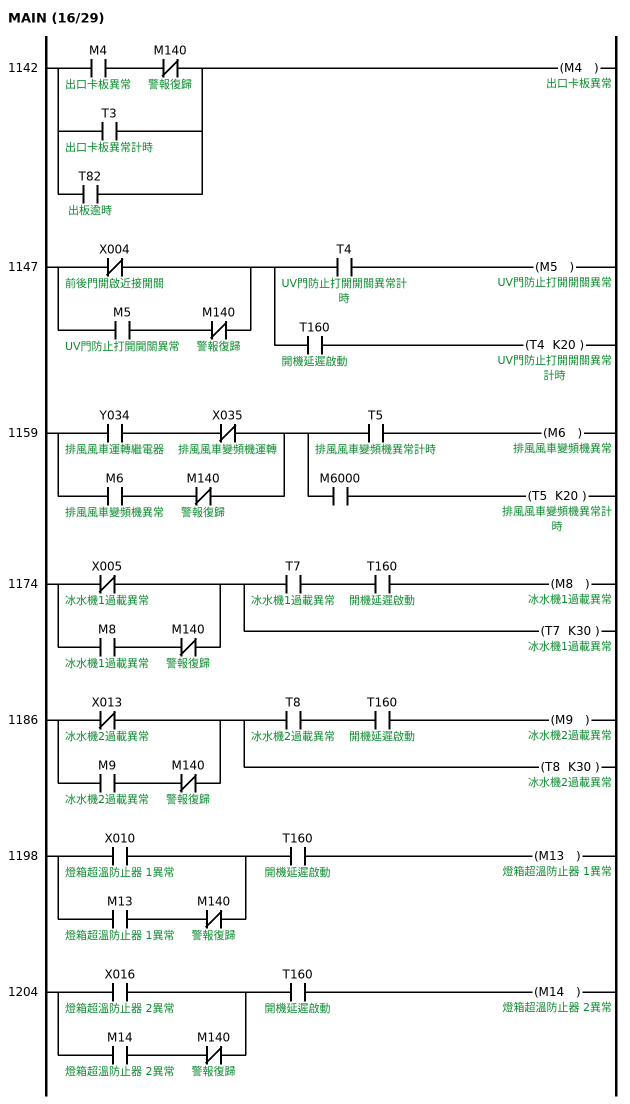
1142  LD      M4  ; 出口卡板異常
      ANI     M140  ; 警報復歸
      OR      T3  ; 出口卡板異常計時
      OR      T82  ; 出板逾時
      OUT     M4  ; 出口卡板異常
1147  LDI     X004  ; 前後門開啟近接開關
      LD      M5  ; UV門防止打開開關異常
      ANI     M140  ; 警報復歸
      ORB
      MPS
      AND     T4  ; UV門防止打開開關異常計時
      OUT     M5  ; UV門防止打開開關異常
      MPP
      AND     T160  ; 開機延遲啟動
      OUT     T4 K20  ; UV門防止打開開關異常計時
1159  LD      Y034  ; 排風風車運轉繼電器
      ANI     X035  ; 排風風車變頻機運轉
      LD      M6  ; 排風風車變頻機異常
      ANI     M140  ; 警報復歸
      ORB
      MPS
      AND     T5  ; 排風風車變頻機異常計時
      OUT     M6  ; 排風風車變頻機異常
      MPP
      AND     M6000
      OUT     T5 K20  ; 排風風車變頻機異常計時
1174  LDI     X005  ; 冰水機1過載異常
      LD      M8  ; 冰水機1過載異常
      ANI     M140  ; 警報復歸
      ORB
      MPS
      AND     T7  ; 冰水機1過載異常
      AND     T160  ; 開機延遲啟動
      OUT     M8  ; 冰水機1過載異常
      MPP
      OUT     T7 K30  ; 冰水機1過載異常
1186  LDI     X013  ; 冰水機2過載異常
      LD      M9  ; 冰水機2過載異常
      ANI     M140  ; 警報復歸
      ORB
      MPS
      AND     T8  ; 冰水機2過載異常
      AND     T160  ; 開機延遲啟動
      OUT     M9  ; 冰水機2過載異常
      MPP
      OUT     T8 K30  ; 冰水機2過載異常
1198  LD      X010  ; 燈箱超溫防止器 1異常
      LD      M13  ; 燈箱超溫防止器 1異常
      ANI     M140  ; 警報復歸
      ORB
      AND     T160  ; 開機延遲啟動
      OUT     M13  ; 燈箱超溫防止器 1異常
1204  LD      X016  ; 燈箱超溫防止器 2異常
      LD      M14  ; 燈箱超溫防止器 2異常
      ANI     M140  ; 警報復歸
      ORB
      AND     T160  ; 開機延遲啟動
      OUT     M14  ; 燈箱超溫防止器 2異常
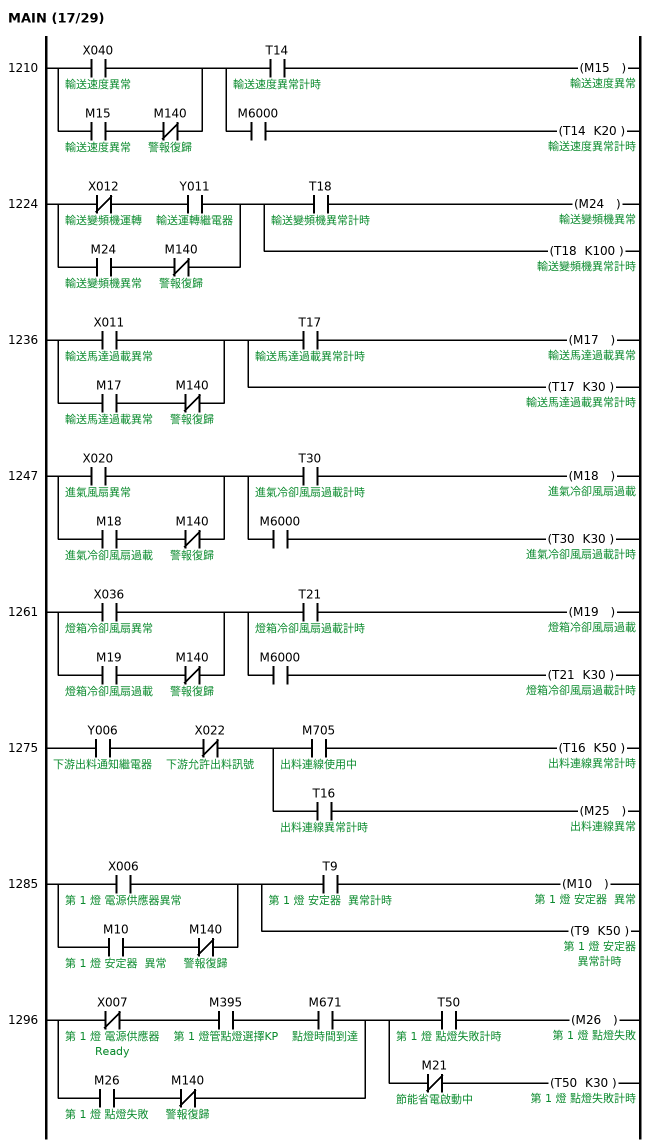
1210  LD      X040  ; 輸送速度異常
      LD      M15  ; 輸送速度異常
      ANI     M140  ; 警報復歸
      ORB
      MPS
      AND     T14  ; 輸送速度異常計時
      OUT     M15  ; 輸送速度異常
      MPP
      AND     M6000
      OUT     T14 K20  ; 輸送速度異常計時
1224  LDI     X012  ; 輸送變頻機運轉
      AND     Y011  ; 輸送運轉繼電器
      LD      M24  ; 輸送變頻機異常
      ANI     M140  ; 警報復歸
      ORB
      MPS
      AND     T18  ; 輸送變頻機異常計時
      OUT     M24  ; 輸送變頻機異常
      MPP
      OUT     T18 K100  ; 輸送變頻機異常計時
1236  LD      X011  ; 輸送馬達過載異常
      LD      M17  ; 輸送馬達過載異常
      ANI     M140  ; 警報復歸
      ORB
      MPS
      AND     T17  ; 輸送馬達過載異常計時
      OUT     M17  ; 輸送馬達過載異常
      MPP
      OUT     T17 K30  ; 輸送馬達過載異常計時
1247  LD      X020  ; 進氣風扇異常
      LD      M18  ; 進氣冷卻風扇過載
      ANI     M140  ; 警報復歸
      ORB
      MPS
      AND     T30  ; 進氣冷卻風扇過載計時
      OUT     M18  ; 進氣冷卻風扇過載
      MPP
      AND     M6000
      OUT     T30 K30  ; 進氣冷卻風扇過載計時
1261  LD      X036  ; 燈箱冷卻風扇異常
      LD      M19  ; 燈箱冷卻風扇過載
      ANI     M140  ; 警報復歸
      ORB
      MPS
      AND     T21  ; 燈箱冷卻風扇過載計時
      OUT     M19  ; 燈箱冷卻風扇過載
      MPP
      AND     M6000
      OUT     T21 K30  ; 燈箱冷卻風扇過載計時
1275  LD      Y006  ; 下游出料通知繼電器
      ANI     X022  ; 下游允許出料訊號
      MPS
      AND     M705  ; 出料連線使用中
      OUT     T16 K50  ; 出料連線異常計時
      MPP
      AND     T16  ; 出料連線異常計時
      OUT     M25  ; 出料連線異常
1285  LD      X006  ; 第 1 燈 電源供應器異常
      LD      M10  ; 第 1 燈 安定器  異常
      ANI     M140  ; 警報復歸
      ORB
      MPS
      AND     T9  ; 第 1 燈 安定器  異常計時
      OUT     M10  ; 第 1 燈 安定器  異常
      MPP
      OUT     T9 K50  ; 第 1 燈 安定器  異常計時
1296  LDI     X007  ; 第 1 燈 電源供應器 Ready
      AND     M395  ; 第 1 燈管點燈選擇KP
      AND     M671  ; 點燈時間到達
      LD      M26  ; 第 1 燈 點燈失敗
      ANI     M140  ; 警報復歸
      ORB
      MPS
      AND     T50  ; 第 1 燈 點燈失敗計時
      OUT     M26  ; 第 1 燈 點燈失敗
      MPP
      ANI     M21  ; 節能省電啟動中
      OUT     T50 K30  ; 第 1 燈 點燈失敗計時
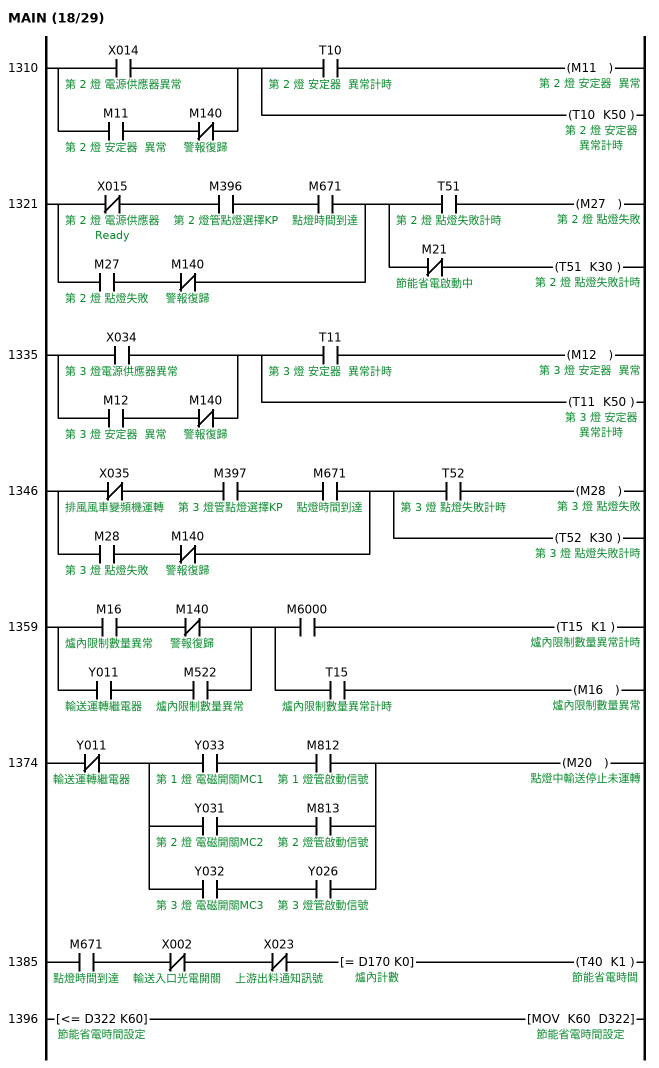
1310  LD      X014  ; 第 2 燈 電源供應器異常
      LD      M11  ; 第 2 燈 安定器  異常
      ANI     M140  ; 警報復歸
      ORB
      MPS
      AND     T10  ; 第 2 燈 安定器  異常計時
      OUT     M11  ; 第 2 燈 安定器  異常
      MPP
      OUT     T10 K50  ; 第 2 燈 安定器  異常計時
1321  LDI     X015  ; 第 2 燈 電源供應器 Ready
      AND     M396  ; 第 2 燈管點燈選擇KP
      AND     M671  ; 點燈時間到達
      LD      M27  ; 第 2 燈 點燈失敗
      ANI     M140  ; 警報復歸
      ORB
      MPS
      AND     T51  ; 第 2 燈 點燈失敗計時
      OUT     M27  ; 第 2 燈 點燈失敗
      MPP
      ANI     M21  ; 節能省電啟動中
      OUT     T51 K30  ; 第 2 燈 點燈失敗計時
1335  LD      X034  ; 第 3 燈電源供應器異常
      LD      M12  ; 第 3 燈 安定器  異常
      ANI     M140  ; 警報復歸
      ORB
      MPS
      AND     T11  ; 第 3 燈 安定器  異常計時
      OUT     M12  ; 第 3 燈 安定器  異常
      MPP
      OUT     T11 K50  ; 第 3 燈 安定器  異常計時
1346  LDI     X035  ; 排風風車變頻機運轉
      AND     M397  ; 第 3 燈管點燈選擇KP
      AND     M671  ; 點燈時間到達
      LD      M28  ; 第 3 燈 點燈失敗
      ANI     M140  ; 警報復歸
      ORB
      MPS
      AND     T52  ; 第 3 燈 點燈失敗計時
      OUT     M28  ; 第 3 燈 點燈失敗
      MPP
      OUT     T52 K30  ; 第 3 燈 點燈失敗計時
1359  LD      M16  ; 爐內限制數量異常
      ANI     M140  ; 警報復歸
      LD      Y011  ; 輸送運轉繼電器
      AND     M522  ; 爐內限制數量異常
      ORB
      MPS
      AND     M6000
      OUT     T15 K1  ; 爐內限制數量異常計時
      MPP
      AND     T15  ; 爐內限制數量異常計時
      OUT     M16  ; 爐內限制數量異常
1374  LDI     Y011  ; 輸送運轉繼電器
      LD      Y033  ; 第 1 燈 電磁開關MC1
      AND     M812  ; 第 1 燈管啟動信號
      LD      Y031  ; 第 2 燈 電磁開關MC2
      AND     M813  ; 第 2 燈管啟動信號
      ORB
      LD      Y032  ; 第 3 燈 電磁開關MC3
      AND     Y026  ; 第 3 燈管啟動信號
      ORB
      ANB
      OUT     M20  ; 點燈中輸送停止未運轉
1385  LD      M671  ; 點燈時間到達
      ANI     X002  ; 輸送入口光電開關
      ANI     X023  ; 上游出料通知訊號
      AND=    D170 K0  ; 爐內計數
      OUT     T40 K1  ; 節能省電時間
1396  LD<=    D322 K60  ; 節能省電時間設定
      MOV     K60 D322
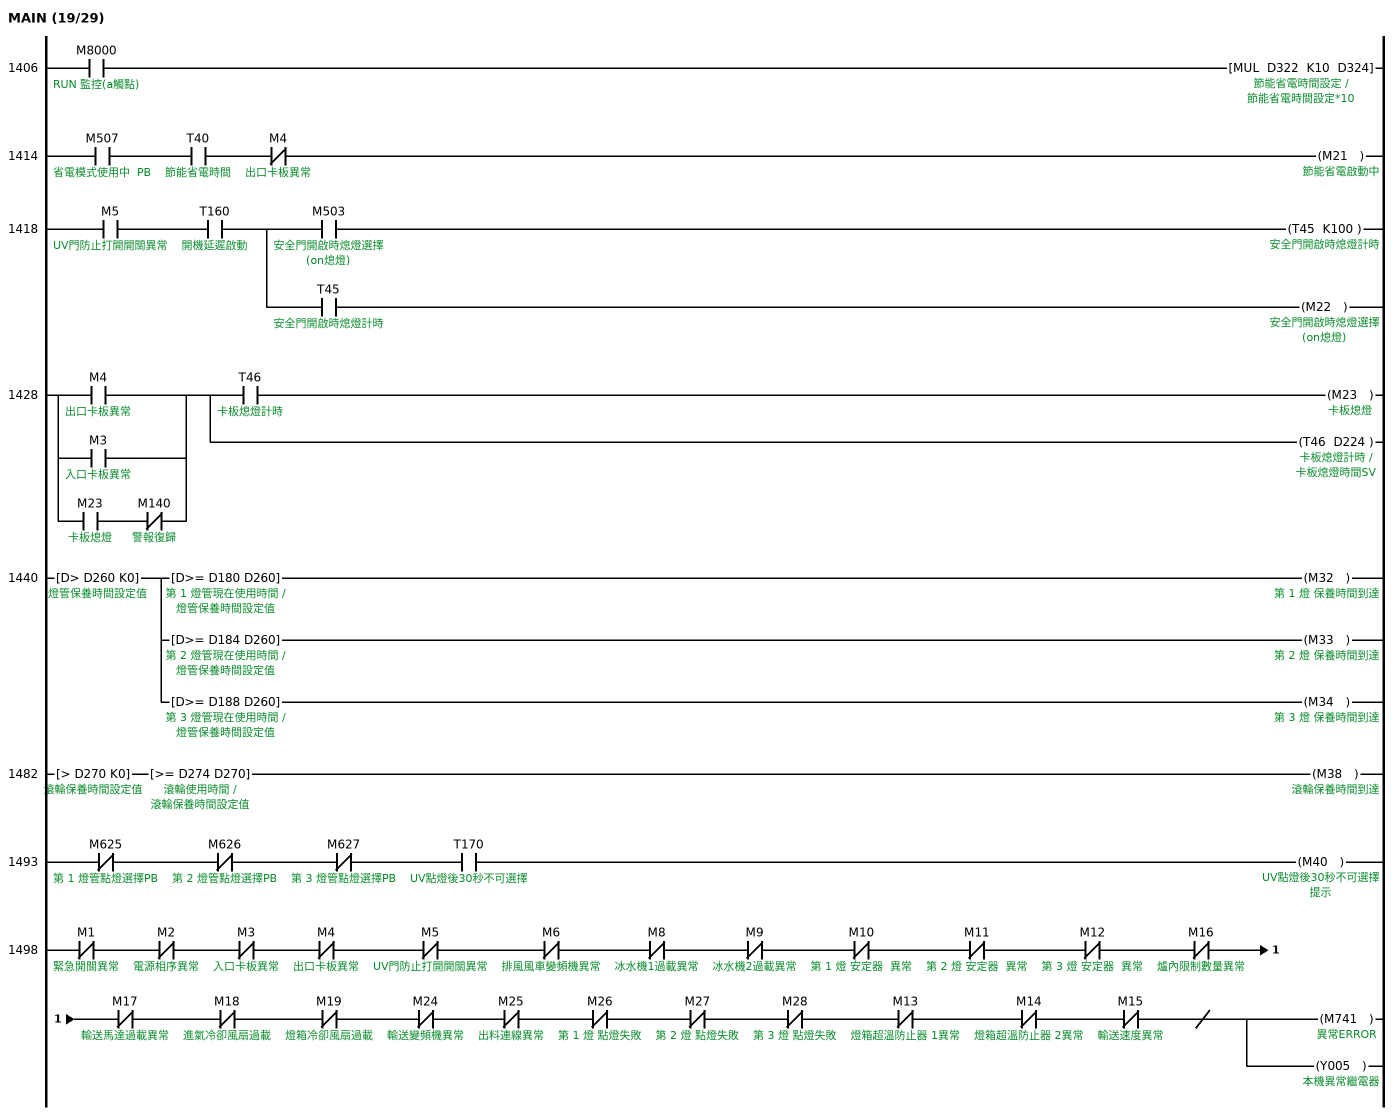
1406  LD      M8000  ; RUN 監控(a觸點)
      MUL     D322 K10 D324  ; 節能省電時間設定*10
1414  LD      M507  ; 省電模式使用中  PB
      AND     T40  ; 節能省電時間
      ANI     M4  ; 出口卡板異常
      OUT     M21  ; 節能省電啟動中
1418  LD      M5  ; UV門防止打開開關異常
      AND     T160  ; 開機延遲啟動
      MPS
      AND     M503  ; 安全門開啟時熄燈選擇    (on熄燈)
      OUT     T45 K100  ; 安全門開啟時熄燈計時
      MPP
      AND     T45  ; 安全門開啟時熄燈計時
      OUT     M22  ; 安全門開啟時熄燈選擇    (on熄燈)
1428  LD      M4  ; 出口卡板異常
      OR      M3  ; 入口卡板異常
      LD      M23  ; 卡板熄燈
      ANI     M140  ; 警報復歸
      ORB
      MPS
      AND     T46  ; 卡板熄燈計時
      OUT     M23  ; 卡板熄燈
      MPP
      OUT     T46 D224  ; 卡板熄燈計時 / 卡板熄燈時間SV
1440  LDD>    D260 K0  ; 燈管保養時間設定值
      MPS
      ANDD>=  D180 D260  ; 第 1 燈管現在使用時間 / 燈管保養時間設定值
      OUT     M32  ; 第 1 燈 保養時間到達
      MRD
      ANDD>=  D184 D260  ; 第 2 燈管現在使用時間 / 燈管保養時間設定值
      OUT     M33  ; 第 2 燈 保養時間到達
      MPP
      ANDD>=  D188 D260  ; 第 3 燈管現在使用時間 / 燈管保養時間設定值
      OUT     M34  ; 第 3 燈 保養時間到達
1482  LD>     D270 K0  ; 滾輪保養時間設定值
      AND>=   D274 D270  ; 滾輪使用時間 / 滾輪保養時間設定值
      OUT     M38  ; 滾輪保養時間到達
1493  LDI     M625  ; 第 1 燈管點燈選擇PB
      ANI     M626  ; 第 2 燈管點燈選擇PB
      ANI     M627  ; 第 3 燈管點燈選擇PB
      AND     T170  ; UV點燈後30秒不可選擇
      OUT     M40  ; UV點燈後30秒不可選擇提示
1498  LDI     M1  ; 緊急開關異常
      ANI     M2  ; 電源相序異常
      ANI     M3  ; 入口卡板異常
      ANI     M4  ; 出口卡板異常
      ANI     M5  ; UV門防止打開開關異常
      ANI     M6  ; 排風風車變頻機異常
      ANI     M8  ; 冰水機1過載異常
      ANI     M9  ; 冰水機2過載異常
      ANI     M10  ; 第 1 燈 安定器  異常
      ANI     M11  ; 第 2 燈 安定器  異常
      ANI     M12  ; 第 3 燈 安定器  異常
      ANI     M16  ; 爐內限制數量異常
      ANI     M17  ; 輸送馬達過載異常
      ANI     M18  ; 進氣冷卻風扇過載
      ANI     M19  ; 燈箱冷卻風扇過載
      ANI     M24  ; 輸送變頻機異常
      ANI     M25  ; 出料連線異常
      ANI     M26  ; 第 1 燈 點燈失敗
      ANI     M27  ; 第 2 燈 點燈失敗
      ANI     M28  ; 第 3 燈 點燈失敗
      ANI     M13  ; 燈箱超溫防止器 1異常
      ANI     M14  ; 燈箱超溫防止器 2異常
      ANI     M15  ; 輸送速度異常
      INV
      OUT     M741  ; 異常ERROR
      OUT     Y005  ; 本機異常繼電器
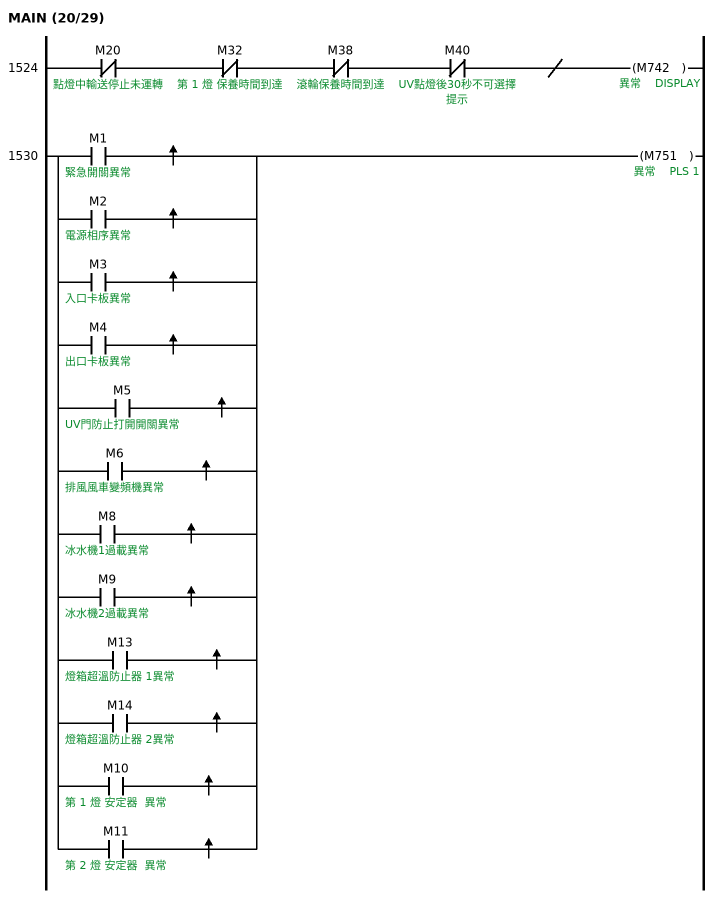
1524  LDI     M20  ; 點燈中輸送停止未運轉
      ANI     M32  ; 第 1 燈 保養時間到達
      ANI     M38  ; 滾輪保養時間到達
      ANI     M40  ; UV點燈後30秒不可選擇提示
      INV
      OUT     M742  ; 異常    DISPLAY
1530  LD      M1  ; 緊急開關異常
      MEP
      LD      M2  ; 電源相序異常
      MEP
      ORB
      LD      M3  ; 入口卡板異常
      MEP
      ORB
      LD      M4  ; 出口卡板異常
      MEP
      ORB
      LD      M5  ; UV門防止打開開關異常
      MEP
      ORB
      LD      M6  ; 排風風車變頻機異常
      MEP
      ORB
      LD      M8  ; 冰水機1過載異常
      MEP
      ORB
      LD      M9  ; 冰水機2過載異常
      MEP
      ORB
      LD      M13  ; 燈箱超溫防止器 1異常
      MEP
      ORB
      LD      M14  ; 燈箱超溫防止器 2異常
      MEP
      ORB
      LD      M10  ; 第 1 燈 安定器  異常
      MEP
      ORB
      LD      M11  ; 第 2 燈 安定器  異常
      MEP
      ORB
      OUT     M751  ; 異常    PLS 1
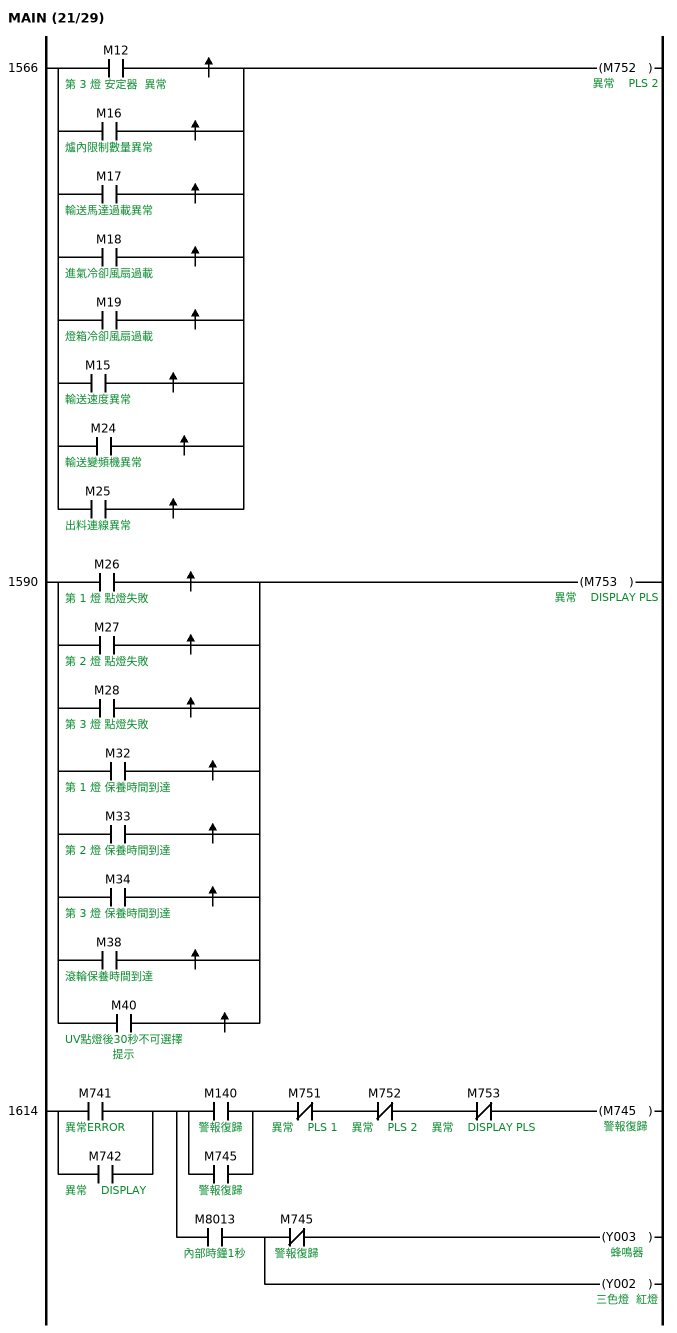
1566  LD      M12  ; 第 3 燈 安定器  異常
      MEP
      LD      M16  ; 爐內限制數量異常
      MEP
      ORB
      LD      M17  ; 輸送馬達過載異常
      MEP
      ORB
      LD      M18  ; 進氣冷卻風扇過載
      MEP
      ORB
      LD      M19  ; 燈箱冷卻風扇過載
      MEP
      ORB
      LD      M15  ; 輸送速度異常
      MEP
      ORB
      LD      M24  ; 輸送變頻機異常
      MEP
      ORB
      LD      M25  ; 出料連線異常
      MEP
      ORB
      OUT     M752  ; 異常    PLS 2
1590  LD      M26  ; 第 1 燈 點燈失敗
      MEP
      LD      M27  ; 第 2 燈 點燈失敗
      MEP
      ORB
      LD      M28  ; 第 3 燈 點燈失敗
      MEP
      ORB
      LD      M32  ; 第 1 燈 保養時間到達
      MEP
      ORB
      LD      M33  ; 第 2 燈 保養時間到達
      MEP
      ORB
      LD      M34  ; 第 3 燈 保養時間到達
      MEP
      ORB
      LD      M38  ; 滾輪保養時間到達
      MEP
      ORB
      LD      M40  ; UV點燈後30秒不可選擇提示
      MEP
      ORB
      OUT     M753  ; 異常    DISPLAY PLS
1614  LD      M741  ; 異常ERROR
      OR      M742  ; 異常    DISPLAY
      MPS
      LD      M140  ; 警報復歸
      OR      M745  ; 警報復歸
      ANB
      ANI     M751  ; 異常    PLS 1
      ANI     M752  ; 異常    PLS 2
      ANI     M753  ; 異常    DISPLAY PLS
      OUT     M745  ; 警報復歸
      MPP
      AND     M8013  ; 內部時鐘1秒
      MPS
      ANI     M745  ; 警報復歸
      OUT     Y003  ; 蜂鳴器
      MPP
      OUT     Y002  ; 三色燈  紅燈
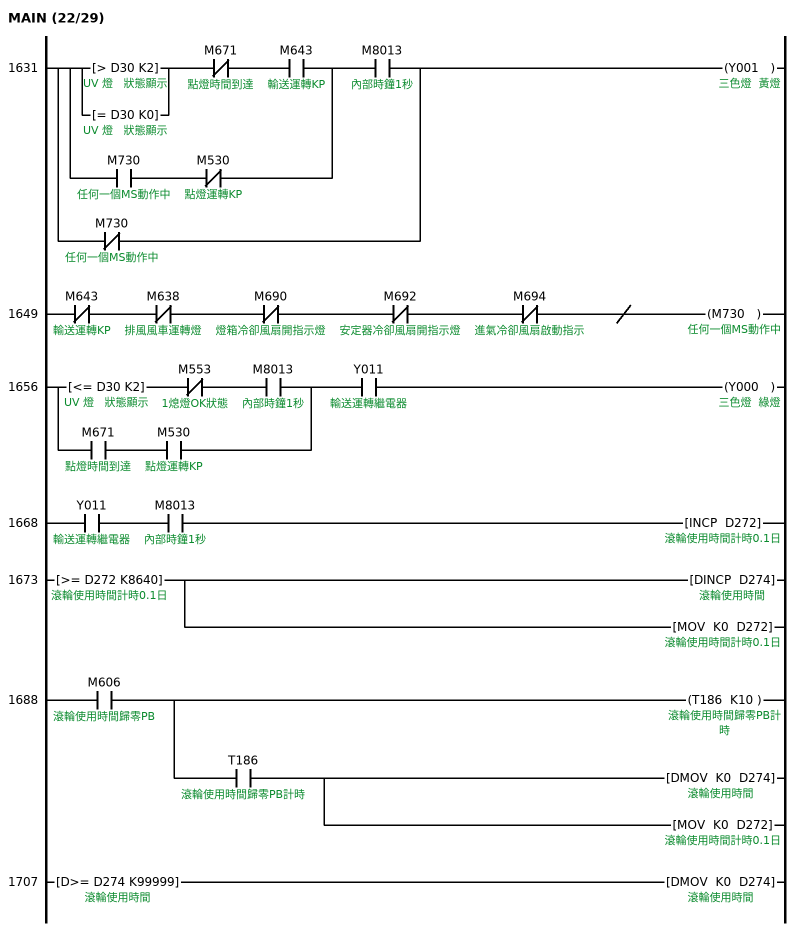
1631  LD>     D30 K2  ; UV 燈   狀態顯示
      OR=     D30 K0  ; UV 燈   狀態顯示
      ANI     M671  ; 點燈時間到達
      AND     M643  ; 輸送運轉KP
      LD      M730  ; 任何一個MS動作中
      ANI     M530  ; 點燈運轉KP
      ORB
      AND     M8013  ; 內部時鐘1秒
      ORI     M730  ; 任何一個MS動作中
      OUT     Y001  ; 三色燈  黃燈
1649  LDI     M643  ; 輸送運轉KP
      ANI     M638  ; 排風風車運轉燈
      ANI     M690  ; 燈箱冷卻風扇開指示燈
      ANI     M692  ; 安定器冷卻風扇開指示燈
      ANI     M694  ; 進氣冷卻風扇啟動指示
      INV
      OUT     M730  ; 任何一個MS動作中
1656  LD<=    D30 K2  ; UV 燈   狀態顯示
      ANI     M553  ; 1熄燈OK狀態
      AND     M8013  ; 內部時鐘1秒
      LD      M671  ; 點燈時間到達
      AND     M530  ; 點燈運轉KP
      ORB
      AND     Y011  ; 輸送運轉繼電器
      OUT     Y000  ; 三色燈  綠燈
1668  LD      Y011  ; 輸送運轉繼電器
      AND     M8013  ; 內部時鐘1秒
      INCP    D272  ; 滾輪使用時間計時0.1日
1673  LD>=    D272 K8640  ; 滾輪使用時間計時0.1日
      DINCP   D274
      MOV     K0 D272
1688  LD      M606  ; 滾輪使用時間歸零PB
      OUT     T186 K10  ; 滾輪使用時間歸零PB計時
      AND     T186  ; 滾輪使用時間歸零PB計時
      DMOV    K0 D274
      MOV     K0 D272
1707  LDD>=   D274 K99999  ; 滾輪使用時間
      DMOV    K0 D274
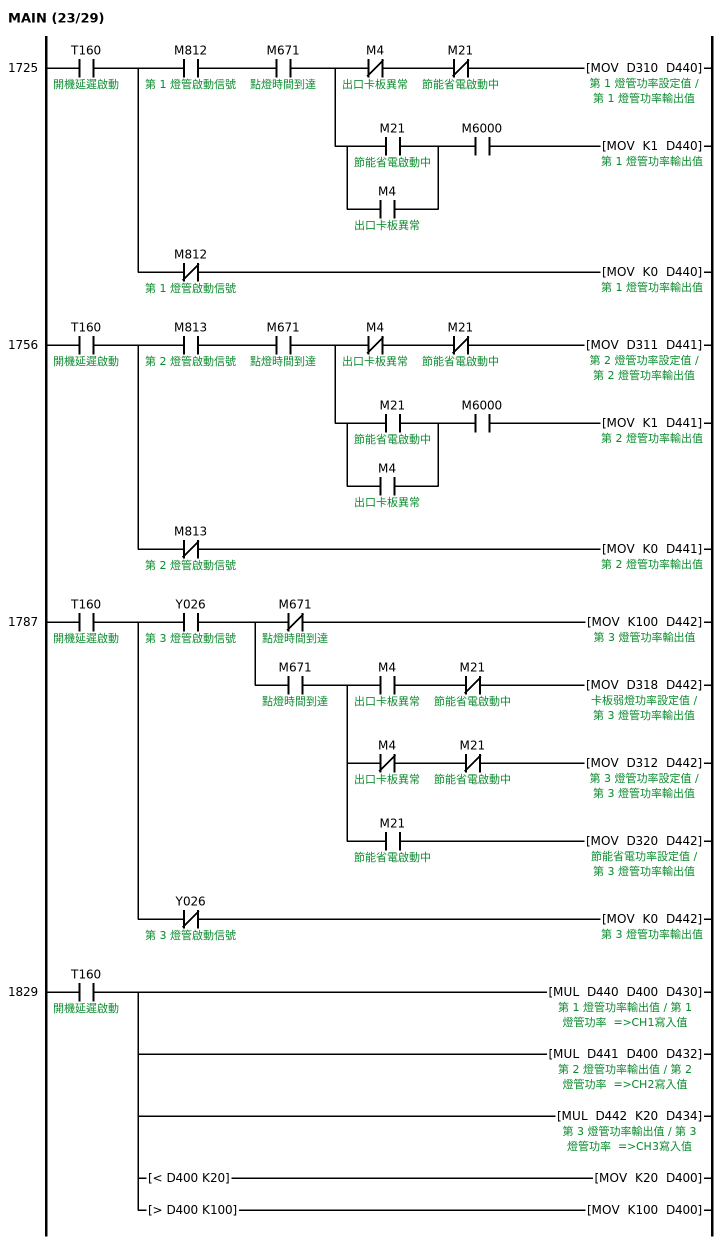
1725  LD      T160  ; 開機延遲啟動
      MPS
      AND     M812  ; 第 1 燈管啟動信號
      AND     M671  ; 點燈時間到達
      MPS
      ANI     M4  ; 出口卡板異常
      ANI     M21  ; 節能省電啟動中
      MOV     D310 D440  ; 第 1 燈管功率輸出值
      MPP
      LD      M21  ; 節能省電啟動中
      OR      M4  ; 出口卡板異常
      ANB
      AND     M6000
      MOV     K1 D440
      MPP
      ANI     M812  ; 第 1 燈管啟動信號
      MOV     K0 D440
1756  LD      T160  ; 開機延遲啟動
      MPS
      AND     M813  ; 第 2 燈管啟動信號
      AND     M671  ; 點燈時間到達
      MPS
      ANI     M4  ; 出口卡板異常
      ANI     M21  ; 節能省電啟動中
      MOV     D311 D441  ; 第 2 燈管功率輸出值
      MPP
      LD      M21  ; 節能省電啟動中
      OR      M4  ; 出口卡板異常
      ANB
      AND     M6000
      MOV     K1 D441
      MPP
      ANI     M813  ; 第 2 燈管啟動信號
      MOV     K0 D441
1787  LD      T160  ; 開機延遲啟動
      MPS
      AND     Y026  ; 第 3 燈管啟動信號
      MPS
      ANI     M671  ; 點燈時間到達
      MOV     K100 D442  ; 第 3 燈管功率輸出值
      MPP
      AND     M671  ; 點燈時間到達
      MPS
      AND     M4  ; 出口卡板異常
      ANI     M21  ; 節能省電啟動中
      MOV     D318 D442
      MRD
      ANI     M4  ; 出口卡板異常
      ANI     M21  ; 節能省電啟動中
      MOV     D312 D442
      MPP
      AND     M21  ; 節能省電啟動中
      MOV     D320 D442
      MPP
      ANI     Y026  ; 第 3 燈管啟動信號
      MOV     K0 D442
1829  LD      T160  ; 開機延遲啟動
      MUL     D440 D400 D430  ; 第 1 燈管功率  =>CH1寫入值
      MUL     D441 D400 D432  ; 第 2 燈管功率  =>CH2寫入值
      MUL     D442 K20 D434  ; 第 3 燈管功率  =>CH3寫入值
      MPS
      AND<    D400 K20
      MOV     K20 D400
      MPP
      AND>    D400 K100
      MOV     K100 D400
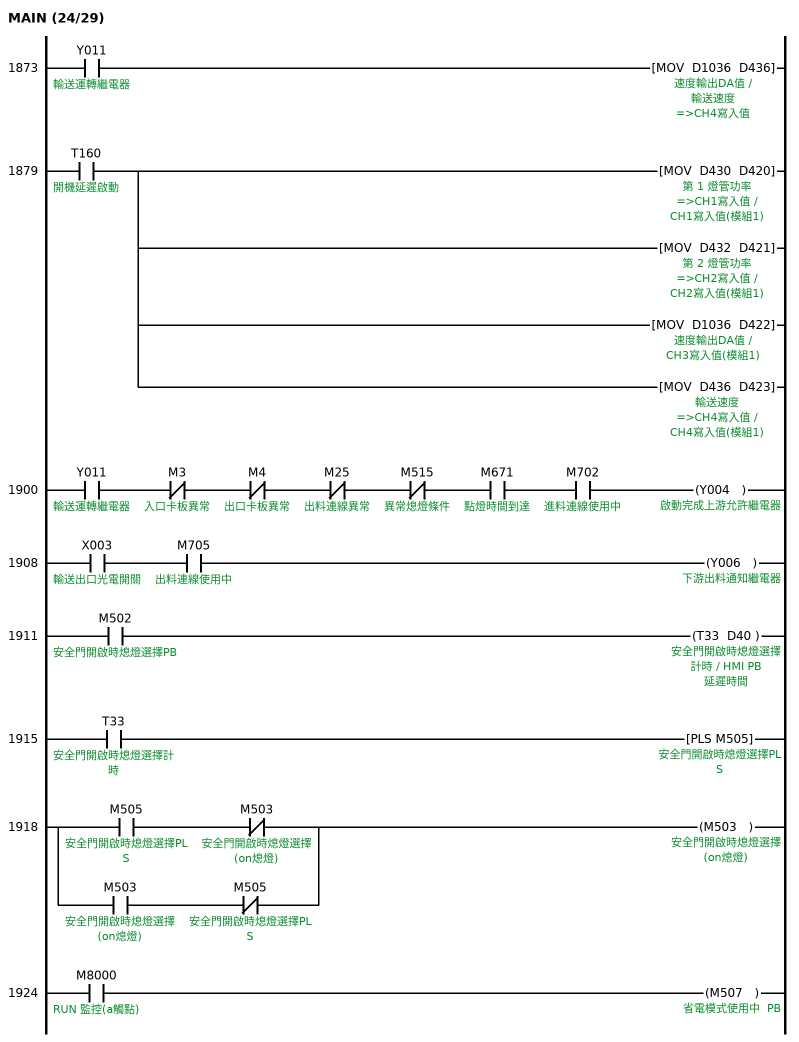
1873  LD      Y011  ; 輸送運轉繼電器
      MOV     D1036 D436  ; 速度輸出DA值 / 輸送速度      =>CH4寫入值
1879  LD      T160  ; 開機延遲啟動
      MOV     D430 D420
      MOV     D432 D421  ; CH2寫入值(模組1)
      MOV     D1036 D422  ; CH3寫入值(模組1)
      MOV     D436 D423  ; CH4寫入值(模組1)
1900  LD      Y011  ; 輸送運轉繼電器
      ANI     M3  ; 入口卡板異常
      ANI     M4  ; 出口卡板異常
      ANI     M25  ; 出料連線異常
      ANI     M515  ; 異常熄燈條件
      AND     M671  ; 點燈時間到達
      AND     M702  ; 進料連線使用中
      OUT     Y004  ; 啟動完成上游允許繼電器
1908  LD      X003  ; 輸送出口光電開關
      AND     M705  ; 出料連線使用中
      OUT     Y006  ; 下游出料通知繼電器
1911  LD      M502  ; 安全門開啟時熄燈選擇PB
      OUT     T33 D40  ; 安全門開啟時熄燈選擇計時 / HMI PB  延遲時間
1915  LD      T33  ; 安全門開啟時熄燈選擇計時
      PLS     M505  ; 安全門開啟時熄燈選擇PLS
1918  LD      M505  ; 安全門開啟時熄燈選擇PLS
      ANI     M503  ; 安全門開啟時熄燈選擇    (on熄燈)
      LD      M503  ; 安全門開啟時熄燈選擇    (on熄燈)
      ANI     M505  ; 安全門開啟時熄燈選擇PLS
      ORB
      OUT     M503  ; 安全門開啟時熄燈選擇    (on熄燈)
1924  LD      M8000  ; RUN 監控(a觸點)
      OUT     M507  ; 省電模式使用中  PB
